METHOD PROTECTED M_DbAlarms : STRING(255)
VAR_INPUT
	nSQLErrorCode				: UDINT;
END_VAR
CASE DatabaseType OF
E_DatabaseType.eMicrosoftSqlCompact,E_DatabaseType.eMicrosoftSql,E_DatabaseType.eMicrosoftAccess:
	CASE nSQLErrorCode OF
		16#80040E00: M_DbAlarms:='Invalid accessor';
		16#80040E01: M_DbAlarms:='Creating another row would have exceeded the total number of active rows supported by the rowset';
		16#80040E02: M_DbAlarms:='Unable to write with a read-only accessor';
		16#80040E03: M_DbAlarms:='Given values violate the database schema';
		16#80040E04: M_DbAlarms:='Invalid row handle';
		16#80040E05: M_DbAlarms:='An object was open';
		16#80040E06: M_DbAlarms:='Invalid chapter';
		16#80040E07: M_DbAlarms:='A literal value in the command could not be converted to the correct type due to a reason other than data overflow';
		16#80040E08: M_DbAlarms:='Invalid binding info';
		16#80040E09: M_DbAlarms:='Permission denied'; 
		16#80040E0A: M_DbAlarms:='Specified column does not contain bookmarks or chapters';
		16#80040E0B: M_DbAlarms:='Some cost limits were rejected';
		16#80040E0C: M_DbAlarms:='No command has been set for the command object';
		16#80040E0D: M_DbAlarms:='Unable to find a query plan within the given cost limit';
		16#80040E0E: M_DbAlarms:='Invalid bookmark';
		16#80040E0F: M_DbAlarms:='Invalid lock mode';
		16#80040E10: M_DbAlarms:='No value given for one or more required parameters';
		16#80040E11: M_DbAlarms:='Invalid column ID';
		16#80040E12: M_DbAlarms:='Invalid ratio';
		16#80040E13: M_DbAlarms:='Invalid value';
		16#80040E14: M_DbAlarms:='The command contained one or more errors';
		16#80040E15: M_DbAlarms:='The executing command cannot be canceled';
		16#80040E16: M_DbAlarms:='The provider does not support the specified dialect';
		16#80040E17: M_DbAlarms:='A data source with the specified name already exists';
		16#80040E18: M_DbAlarms:='The rowset was builtover a live data feed and cannot be restarted';
		16#80040E19: M_DbAlarms:='No key matching the described characteristics could be found within the current range';
		16#80040E1A: M_DbAlarms:='Ownership of this tree has been given to the provider';
		16#80040E1B: M_DbAlarms:='The provider is unable to determine identity for newly inserted rows';
		16#80040E1C: M_DbAlarms:='No nonzero weights specified for any goals supported, so goal was rejected; current goal was not changed';
		16#80040E1D: M_DbAlarms:='Requested conversion is not supported';
		16#80040E1E: M_DbAlarms:='lRowsOffset would position you past either end of the rowset, regardless of the cRows value specified; cRowsObtained is 0';
		16#80040E1F: M_DbAlarms:='Information was requested for a query, and the query was not set';
		16#80040E20: M_DbAlarms:='Provider called a method from IRowsetNotify in the consumer and NT';
		16#80040E21: M_DbAlarms:='Errors occurred';
		16#80040E22: M_DbAlarms:='A non-NULL controlling IUnknown was specified and the object being created does not support aggregation';
		16#80040E23: M_DbAlarms:='A given HROW referred to a hard- or soft-deleted row';
		16#80040E24: M_DbAlarms:='The rowset does not support fetching backwards';
		16#80040E25: M_DbAlarms:='All HROWs must be released before new ones can be obtained';
		16#80040E26: M_DbAlarms:='One of the specified storage flags was not supported';
		16#80040E27: M_DbAlarms:='The comparison operator was invalid';
		16#80040E28: M_DbAlarms:='The specified status flag was neither DBCOLUMNSTATUS_OK nor DBCOLUMNSTATUS_ISNUL';
		16#80040E29: M_DbAlarms:='The rowset cannot scroll backwards';
		16#80040E2A: M_DbAlarms:='Invalid region handle';
		16#80040E2B: M_DbAlarms:='The specified set of rows was not contiguous to or overlapping the rows in the specified watch region';
		16#80040E2C: M_DbAlarms:='A transition from ALL* to MOVE* or EXTEND* was specified';
		16#80040E2D: M_DbAlarms:='The specified region is not a proper subregion of the region identified by the given watch region handle';
		16#80040E2E: M_DbAlarms:='The provider does not support multi-statement commands';
		16#80040E2F: M_DbAlarms:='A specified value violated the integrity constraints for a column or table';
		16#80040E30: M_DbAlarms:='The given type name was unrecognized';
		16#80040E31: M_DbAlarms:='Execution aborted because a resource limit has been reached; no results have been returned';
		16#80040E32: M_DbAlarms:='Cannot clone a command object whose command tree contains a rowset or rowsets';
		16#80040E33: M_DbAlarms:='Cannot represent the current tree as text';
		16#80040E34: M_DbAlarms:='The specified index already exists';
		16#80040E35: M_DbAlarms:='The specified index does not exist';
		16#80040E36: M_DbAlarms:='The specified index was in use';
		16#80040E37: M_DbAlarms:='The specified table does not exist';
		16#80040E38: M_DbAlarms:='The rowset was using optimistic concurrency and the value of a column has been changed since it was last read';
		16#80040E39: M_DbAlarms:='Errors were detected during the copy';
		16#80040E3A: M_DbAlarms:='A specified precision was invalid';
		16#80040E3B: M_DbAlarms:='A specified scale was invalid';
		16#80040E3C: M_DbAlarms:='Invalid table ID';
		16#80040E3D: M_DbAlarms:='A specified type was invalid';
		16#80040E3E: M_DbAlarms:='A column ID was occurred more than once in the specification';
		16#80040E3F: M_DbAlarms:='The specified table already exists';
		16#80040E40: M_DbAlarms:='The specified table was in use';
		16#80040E41: M_DbAlarms:='The specified locale ID was not supported';
		16#80040E42: M_DbAlarms:='The specified record number is invalid';
		16#80040E43: M_DbAlarms:='Although the bookmark was validly formed, no row could be found to match it';
		16#80040E44: M_DbAlarms:='The value of a property was invalid';
		16#80040E45: M_DbAlarms:='The rowset was not chaptered';
		16#80040E46: M_DbAlarms:='Invalid accessor';
		16#80040E47: M_DbAlarms:='Invalid storage flags';
		16#80040E48: M_DbAlarms:='By-ref accessors are not supported by this provider';
		16#80040E49: M_DbAlarms:='Null accessors are not supported by this provider';
		16#80040E4A: M_DbAlarms:='The command was not prepared';
		16#80040E4B: M_DbAlarms:='The specified accessor was not a parameter accessor';
		16#80040E4C: M_DbAlarms:='The given accessor was write-only';
		16#80040E4D: M_DbAlarms:='Authentication failed';
		16#80040E4E: M_DbAlarms:='The change was canceled during notification; no columns are changed';
		16#80040E4F: M_DbAlarms:='The rowset was single-chaptered and the chapter was not released';
		16#80040E50: M_DbAlarms:='Invalid source handle';
		16#80040E51: M_DbAlarms:='The provider cannot derive parameter info and SetParameterInfo has not been called';
		16#80040E52: M_DbAlarms:='The data source object is already initialized';
		16#80040E53: M_DbAlarms:='The provider does not support this method';
		16#80040E54: M_DbAlarms:='The number of rows with pending changes has exceeded the set limit';
		16#80040E55: M_DbAlarms:='The specified column did not exist';
		16#80040E56: M_DbAlarms:='There are pending changes on a row with a reference count of zero';
		16#80040E57: M_DbAlarms:='A literal value in the command overflowed the range of the type of the associated column';
		16#80040E58: M_DbAlarms:='The supplied HRESULT was invalid';
		16#80040E59: M_DbAlarms:='The supplied LookupID was invalid';
		16#80040E5A: M_DbAlarms:='The supplied DynamicErrorID was invalid';
		16#80040E5B: M_DbAlarms:='Unable to get visible data for a newly-inserted row that has not yet been updated';
		16#80040E5C: M_DbAlarms:='Invalid conversion flag';
		16#80040E5D: M_DbAlarms:='The given parameter name was unrecognized';
		16#80040E5E: M_DbAlarms:='Multiple storage objects can not be open simultaneously';
		16#80040E5F: M_DbAlarms:='The requested filter could not be opened';
		16#80040E60: M_DbAlarms:='The requested order could not be opened';
		16#80040E61: M_DbAlarms:='Bad tuple';
		16#80040E62: M_DbAlarms:='Bad coordinate';
		16#80040E63: M_DbAlarms:='The given axis was not valid for this Dataset';
		16#80040E64: M_DbAlarms:='One or more of the given cell ordinals was invalid';
		16#80040E65: M_DbAlarms:='The supplied columnID was invalid';
		16#80040E67: M_DbAlarms:='The supplied command does not have a DBID (Note: DBID is SQL shorthand for Database ID.)';
		16#80040E68: M_DbAlarms:='The supplied DBID already exists';
		16#80040E69: M_DbAlarms:='The maximum number of Sessions supported by the provider has already been created. The consumer must release one or more currently held Sessions before obtaining a new Session object';
		16#80040E72: M_DbAlarms:='The index ID is invalid';
		16#80040E73: M_DbAlarms:='The initialization string does not conform to specification';
		16#80040E74: M_DbAlarms:='The OLE DB root enumerator did not return any providers that matched an of the SOURCES_TYPEs requested';
		16#80040E75: M_DbAlarms:='The initialization string specifies a provider which does not match the currently active provider.';
		16#80040E76: M_DbAlarms:='The specified DBID is invalid';
		16#80040E6A: M_DbAlarms:='Invalid trustee value';
		16#80040E6B: M_DbAlarms:='The trustee is not for the current data source';
		16#80040E6C: M_DbAlarms:='The trustee does not support memberships/collections';
		16#80040E6D: M_DbAlarms:='The object is invalid or unknown to the provider';
		16#80040E6E: M_DbAlarms:='No owner exists for the object';
		16#80040E6F: M_DbAlarms:='The access entry list supplied is invalid';
		16#80040E70: M_DbAlarms:='The trustee supplied as owner is invalid or unknown to the provider';
		16#80040E71: M_DbAlarms:='The permission supplied in the access entry list is invalid';
		16#80040E77: M_DbAlarms:='The ConstraintType was invalid or not supported by the provider.';
		16#80040E78: M_DbAlarms:='The ConstraintType was not CONSTRAINTTYPE_FOREIGNKEY and cForeignKeyColumns was not zero';
		16#80040E79: M_DbAlarms:='The Deferrability was invalid or the value was not supported by the provider';
		16#80040E80: M_DbAlarms:='The MatchType was invalid or the value was not supported by the provider';
		16#80040E8A: M_DbAlarms:='The UpdateRule or DeleteRule was invalid or the value was not supported by the provider';
		16#80040E8B: M_DbAlarms:='The pConstraintID did not exist in the data source';
		16#80040E8C: M_DbAlarms:='The dwFlags was invalid';
		16#80040E8D: M_DbAlarms:='The rguidColumnType pointed to a GUID that does not match the object type of this column or this column was not set';
		16#80040E8E: M_DbAlarms:='The requested URL was out-of-scope';
		16#80040E90: M_DbAlarms:='The provider could not drop the object';
		16#80040E91: M_DbAlarms:='There is no source row';
		16#80040E92: M_DbAlarms:='The OLE DB object represented by this URL is locked by one or more other processes';
		16#80040E93: M_DbAlarms:='The client requested an object type that is only valid for a collection';
		16#80040E94: M_DbAlarms:='The caller requested write access to a read-only object';
		16#80040E95: M_DbAlarms:='The provider could not connect to the server for this object';
		16#80040E96: M_DbAlarms:='The provider could not connect to the server for this object';
		16#80040E97: M_DbAlarms:='The attempt to bind to the object timed out';
		16#80040E98: M_DbAlarms:='The provider was unable to create an object at this URL because an object named by this URL already exists';
		16#80040E99: M_DbAlarms:='The provider could not drop the object';
		16#80040E9A: M_DbAlarms:='The provider was unable to create an object at this URL because the server was out of physical storage';
		16#00040EC0: M_DbAlarms:='Fetching requested number of rows would have exceeded total number of active rows supported by the rowset';
		16#00040EC1: M_DbAlarms:='One or more column types are incompatible; conversion errors will occur during copying';
		16#00040EC2: M_DbAlarms:='Parameter type information has been overridden by caller';
		16#00040EC3: M_DbAlarms:='Skipped bookmark for deleted or non-member row';
		16#00040EC4: M_DbAlarms:='Errors found in validating tree';
		16#00040EC5: M_DbAlarms:='There are no more rowsets';
		16#00040EC6: M_DbAlarms:='Reached start or end of rowset or chapter';
		16#00040EC7: M_DbAlarms:='The provider re-executed the command';
		16#00040EC8: M_DbAlarms:='Variable data buffer ful';
		16#00040EC9: M_DbAlarms:='There are no more results';
		16#00040ECA: M_DbAlarms:='Server cannot release or downgrade a lock until the end of the transaction';
		16#00040ECB: M_DbAlarms:='Specified weight was not supported or exceeded the supported limit and was set to 0 or the supported limit';
		16#00040ECC: M_DbAlarms:='Consumer is uninterested in receiving further notification calls for this reason';
		16#00040ECD: M_DbAlarms:='Input dialect was ignored and text was returned in different dialect';
		16#00040ECE: M_DbAlarms:='Consumer is uninterested in receiving further notification calls for this phase';
		16#00040ECF: M_DbAlarms:='Consumer is uninterested in receiving further notification calls for this reason';
		16#00040ED0: M_DbAlarms:='The operation is being processed asynchronously';
		16#00040ED1: M_DbAlarms:='In order to reposition to the start of the rowset, the provider had to reexecute the query; either the order of the columns changed or columns were added to or removed from the rowset';
		16#00040ED2: M_DbAlarms:='The method had some errors; errors have been returned in the error array';
		16#00040ED3: M_DbAlarms:='Invalid row handle';
		16#00040ED4: M_DbAlarms:='A given HROW referred to a hard-deleted row';
		16#00040ED5: M_DbAlarms:='The provider was unable to keep track of all the changes; the client must refetch the data associated with the watch region using another method';
		16#00040ED6: M_DbAlarms:='Execution stopped because a resource LIMIT has been reached; results obtained so far have been returned but execution cannot be resumed';
		16#00040ED7: M_DbAlarms:='The bind failed because the provider was unable to satisfy all of the bind flags or properties';
		16#00040ED8: M_DbAlarms:='A lock was upgraded FROM the value specified';
		16#00040ED9: M_DbAlarms:='One OR more properties were changed as allowed BY provider';
		16#00040EDA: M_DbAlarms:='Errors occurred';
		16#00040EDB: M_DbAlarms:='A specified parameter was invalid';
		16#00040EDC: M_DbAlarms:='Updating this row caused more than one row to be updated in the data source';
		16#00040EDD: M_DbAlarms:='The row has no row-specific columns';
	ELSE
		M_DbAlarms:= 'Undefined Microsoft Sql Alarm';
	END_CASE
E_DatabaseType.eMySQL:
	//TODO
E_DatabaseType.eOracle:
	//TODO
E_DatabaseType.eDB2:
	//TODO
E_DatabaseType.ePostgreSQL:
	//TODO
E_DatabaseType.eInterbase:
	//TODO
E_DatabaseType.eXml:
	CASE nSQLErrorCode OF
		1:	M_DbAlarms:='FUNCTION NOT allowed.';
		2:	M_DbAlarms:='XML file could not be read';
		3:	M_DbAlarms:='XML schema could not be read';
		4:	M_DbAlarms:='Syntax error';
		5:	M_DbAlarms:='Table could not be created.';
		6:	M_DbAlarms:='The list OF INSERT VALUES are NOT conform TO the collumn list';
		7:	M_DbAlarms:='Memory OF the PLC structure NOT big enough.';
		8:	M_DbAlarms:='XML file could not be created.';
		9:	M_DbAlarms:='XML database not found.';
		10:	M_DbAlarms:='XML table NOT found.';
	ELSE
		M_DbAlarms:= 'Undefined XML DB Alarm';
	END_CASE
E_DatabaseType.eAscii:
	CASE nSQLErrorCode OF
		1:	M_DbAlarms:='FUNCTION NOT allowed.';
		2:	M_DbAlarms:='Syntax error';
		3:	M_DbAlarms:='File could not be open.';
	ELSE
		M_DbAlarms:= 'Undefined ASCII DB Alarm';
	END_CASE
END_CASE
END_METHOD

METHOD PROTECTED M_DbServerAlarms : STRING
VAR_INPUT
	nErrID				: UDINT;
END_VAR
CASE nErrID OF
	131073: M_DbServerAlarms := 'Microsoft SQL Compact database';
	262145: M_DbServerAlarms := 'Microsoft SQL database';
	524289: M_DbServerAlarms := 'Microsoft Access database';
	1048577: M_DbServerAlarms := 'MySQL database';
	2097153: M_DbServerAlarms := 'Oracle database';
	4194305: M_DbServerAlarms := 'DB2 database';
	8388609: M_DbServerAlarms := 'PostgreSQL database';
	16777217: M_DbServerAlarms := 'Interbase/Firebird database';
	33554433: M_DbServerAlarms := 'NULL values are not allowed';
	33554434: M_DbServerAlarms := 'FB_DBRead selected value is NULL';
	33554435: M_DbServerAlarms := 'DBID is unknown';
	33554436: M_DbServerAlarms := 'ADSDevID is unknown';
	33554437: M_DbServerAlarms := 'No open database connection found for DBID xy';
	33554438: M_DbServerAlarms := 'No open ADS device connection found for ADSDevID xy';
	67108865: M_DbServerAlarms := 'XML database';
	134217729: M_DbServerAlarms := 	'ASCII database';
ELSE
	M_DbServerAlarms := 	'ADS Error';
END_CASE
END_METHOD

METHOD PROTECTED M_OdbcAlarms : STRING
VAR_INPUT
	sSQLState    : STRING(5);
END_VAR
IF sSQLState = '1000' THEN  M_OdbcAlarms:= 'General warning';
ELSIF sSQLState ='1001'	THEN M_OdbcAlarms:= 'Cursor operation conflict';
ELSIF sSQLState ='1002'	THEN M_OdbcAlarms:= 'Disconnect error';
ELSIF sSQLState ='1003'	THEN M_OdbcAlarms:= 'NULL value eliminated in set FUNCTION';
ELSIF sSQLState ='1004'	THEN M_OdbcAlarms:= 'STRING data, right-truncated';
ELSIF sSQLState ='1006'	THEN M_OdbcAlarms:= 'Privilege NOT revoked';
ELSIF sSQLState ='1007'	THEN M_OdbcAlarms:= 'Privilege NOT granted';
ELSIF sSQLState ='01S00' THEN M_OdbcAlarms:= 'Invalid connection STRING attribute';
ELSIF sSQLState ='01S01' THEN M_OdbcAlarms:= 'Error in row';
ELSIF sSQLState ='01S02' THEN M_OdbcAlarms:= 'Option value changed';
ELSIF sSQLState ='01S06' THEN M_OdbcAlarms:= 'Attempt TO fetch before the result set returned the first rowset';
ELSIF sSQLState ='01S07' THEN M_OdbcAlarms:= 'Fractional truncation';
ELSIF sSQLState ='01S08' THEN M_OdbcAlarms:= 'Error saving File DSN';
ELSIF sSQLState ='01S09' THEN M_OdbcAlarms:= 'Invalid keyword';
ELSIF sSQLState ='7001'	THEN M_OdbcAlarms:= 'Wrong number OF parameters';
ELSIF sSQLState ='7002'	THEN M_OdbcAlarms:= 'COUNT field incorrect';
ELSIF sSQLState ='7005'	THEN M_OdbcAlarms:= 'Prepared statement not a cursor-specification';
ELSIF sSQLState ='7006'	THEN M_OdbcAlarms:= 'Restricted data type attribute violation';
ELSIF sSQLState ='7009'	THEN M_OdbcAlarms:= 'Invalid descriptor index';
ELSIF sSQLState ='07S01' THEN M_OdbcAlarms:= 'Invalid use OF default parameter';
ELSIF sSQLState ='8001'	THEN M_OdbcAlarms:= 'Client unable TO establish connection';
ELSIF sSQLState ='8002'	THEN M_OdbcAlarms:= 'Connection name in use';
ELSIF sSQLState ='8003'	THEN M_OdbcAlarms:= 'Connection not open';
ELSIF sSQLState ='8004'	THEN M_OdbcAlarms:= 'Server rejected the connection';
ELSIF sSQLState ='8007'	THEN M_OdbcAlarms:= 'Connection failure during transaction';
ELSIF sSQLState ='08S01' THEN M_OdbcAlarms:= 'Communication link failure';
ELSIF sSQLState ='21S01' THEN M_OdbcAlarms:= 'Insert value list does not match column list';
ELSIF sSQLState ='21S02' THEN M_OdbcAlarms:= 'Degree of derived table does not match column list';
ELSIF sSQLState ='22001' THEN M_OdbcAlarms:= 'String data, right-truncated';
ELSIF sSQLState ='22002' THEN M_OdbcAlarms:= 'Indicator variable required but not supplied';
ELSIF sSQLState ='22003' THEN M_OdbcAlarms:= 'Numeric value out of range';
ELSIF sSQLState ='22007' THEN M_OdbcAlarms:= 'Invalid datetime format';
ELSIF sSQLState ='22008' THEN M_OdbcAlarms:= 'Datetime field overflow';
ELSIF sSQLState ='22012' THEN M_OdbcAlarms:= 'Division by zero';
ELSIF sSQLState ='22015' THEN M_OdbcAlarms:= 'Interval field overflow';
ELSIF sSQLState ='22018' THEN M_OdbcAlarms:= 'Invalid character value for cast specification';
ELSIF sSQLState ='22019' THEN M_OdbcAlarms:= 'Invalid escape character';
ELSIF sSQLState ='22025' THEN M_OdbcAlarms:= 'Invalid escape sequence';
ELSIF sSQLState ='22026' THEN M_OdbcAlarms:= 'String data, length mismatch';
ELSIF sSQLState ='23000' THEN M_OdbcAlarms:= 'Integrity constraint violation';
ELSIF sSQLState ='24000' THEN M_OdbcAlarms:= 'Invalid cursor state';
ELSIF sSQLState ='25000' THEN M_OdbcAlarms:= 'Invalid transaction state';
ELSIF sSQLState ='25S01' THEN M_OdbcAlarms:= 'Transaction state';
ELSIF sSQLState ='25S02' THEN M_OdbcAlarms:= 'Transaction is still active';
ELSIF sSQLState ='25S03' THEN M_OdbcAlarms:= 'Transaction is rolled back';
ELSIF sSQLState ='28000' THEN M_OdbcAlarms:= 'Invalid authorization specification';
ELSIF sSQLState ='34000' THEN M_OdbcAlarms:= 'Invalid cursor name';
ELSIF sSQLState ='3C000' THEN M_OdbcAlarms:= 'Duplicate cursor name';
ELSIF sSQLState ='3D000' THEN M_OdbcAlarms:= 'Invalid catalog name';
ELSIF sSQLState ='3F000' THEN M_OdbcAlarms:= 'Invalid schema name';
ELSIF sSQLState ='40001' THEN M_OdbcAlarms:= 'Serialization failure';
ELSIF sSQLState ='40002' THEN M_OdbcAlarms:= 'Integrity constraint violation';
ELSIF sSQLState ='40003' THEN M_OdbcAlarms:= 'Statement completion unknown';
ELSIF sSQLState ='42000' THEN M_OdbcAlarms:= 'Syntax error or access violation';
ELSIF sSQLState ='42S01' THEN M_OdbcAlarms:= 'Base table or view already exists';
ELSIF sSQLState ='42S02' THEN M_OdbcAlarms:= 'Base table or view not found';
ELSIF sSQLState ='42S11' THEN M_OdbcAlarms:= 'Index already exists';
ELSIF sSQLState ='42S12' THEN M_OdbcAlarms:= 'Index not found';
ELSIF sSQLState ='42S21' THEN M_OdbcAlarms:= 'Column already exists';
ELSIF sSQLState ='42S22' THEN M_OdbcAlarms:= 'Column not found';
ELSIF sSQLState ='44000' THEN M_OdbcAlarms:= 'WITH CHECK OPTION violation';
ELSIF sSQLState ='HY000' THEN M_OdbcAlarms:= 'General error';
ELSIF sSQLState ='HY001' THEN M_OdbcAlarms:= 'Memory allocation error';
ELSIF sSQLState ='HY003' THEN M_OdbcAlarms:= 'Invalid application buffer type';
ELSIF sSQLState ='HY004' THEN M_OdbcAlarms:= 'Invalid SQL data type';
ELSIF sSQLState ='HY007' THEN M_OdbcAlarms:= 'Associated statement is not prepared';
ELSIF sSQLState ='HY008' THEN M_OdbcAlarms:= 'Operation canceled';
ELSIF sSQLState ='HY009' THEN M_OdbcAlarms:= 'Invalid use of null pointer';
ELSIF sSQLState ='HY010' THEN M_OdbcAlarms:= 'Function sequence error';
ELSIF sSQLState ='HY011' THEN M_OdbcAlarms:= 'Attribute cannot be set now';
ELSIF sSQLState ='HY012' THEN M_OdbcAlarms:= 'Invalid transaction operation code';
ELSIF sSQLState ='HY013' THEN M_OdbcAlarms:= 'Memory management error';
ELSIF sSQLState ='HY014' THEN M_OdbcAlarms:= 'Limit on the number of handles exceeded';
ELSIF sSQLState ='HY015' THEN M_OdbcAlarms:= 'No cursor name available';
ELSIF sSQLState ='HY016' THEN M_OdbcAlarms:= 'Cannot modify an implementation row descriptor';
ELSIF sSQLState ='HY017' THEN M_OdbcAlarms:= 'Invalid use of an automatically allocated descriptor handle';
ELSIF sSQLState ='HY018' THEN M_OdbcAlarms:= 'Server declined cancel request';
ELSIF sSQLState ='HY019' THEN M_OdbcAlarms:= 'Non-character and non-binary data sent in pieces';
ELSIF sSQLState ='HY020' THEN M_OdbcAlarms:= 'Attempt to concatenate a null value';
ELSIF sSQLState ='HY021' THEN M_OdbcAlarms:= 'Inconsistent descriptor information';
ELSIF sSQLState ='HY024' THEN M_OdbcAlarms:= 'Invalid attribute value';
ELSIF sSQLState ='HY090' THEN M_OdbcAlarms:= 'Invalid string or buffer length';
ELSIF sSQLState ='HY091' THEN M_OdbcAlarms:= 'Invalid descriptor field identifier';
ELSIF sSQLState ='HY092' THEN M_OdbcAlarms:= 'Invalid attribute/option identifier';
ELSIF sSQLState ='HY095' THEN M_OdbcAlarms:= 'Function type out of range';
ELSIF sSQLState ='HY096' THEN M_OdbcAlarms:= 'Invalid information type';
ELSIF sSQLState ='HY097' THEN M_OdbcAlarms:= 'Column type out of range';
ELSIF sSQLState ='HY098' THEN M_OdbcAlarms:= 'Scope type out of range';
ELSIF sSQLState ='HY099' THEN M_OdbcAlarms:= 'Nullable type out of range';
ELSIF sSQLState ='HY100' THEN M_OdbcAlarms:= 'Uniqueness option type out of range';
ELSIF sSQLState ='HY101' THEN M_OdbcAlarms:= 'Accuracy option type out of range';
ELSIF sSQLState ='HY103' THEN M_OdbcAlarms:= 'Invalid retrieval code';
ELSIF sSQLState ='HY104' THEN M_OdbcAlarms:= 'Invalid precision or scale value';
ELSIF sSQLState ='HY105' THEN M_OdbcAlarms:= 'Invalid parameter type';
ELSIF sSQLState ='HY106' THEN M_OdbcAlarms:= 'Fetch type out of range';
ELSIF sSQLState ='HY107' THEN M_OdbcAlarms:= 'Row value out of range';
ELSIF sSQLState ='HY109' THEN M_OdbcAlarms:= 'Invalid cursor position';
ELSIF sSQLState ='HY110' THEN M_OdbcAlarms:= 'Invalid driver completion';
ELSIF sSQLState ='HY111' THEN M_OdbcAlarms:= 'Invalid bookmark value';
ELSIF sSQLState ='HYC00' THEN M_OdbcAlarms:= 'Optional feature not implemented';
ELSIF sSQLState ='HYT00' THEN M_OdbcAlarms:= 'Timeout expired';
ELSIF sSQLState ='HYT01' THEN M_OdbcAlarms:= 'Connection timeout expired';
ELSIF sSQLState ='IM001' THEN M_OdbcAlarms:= 'Driver does not support this function';
ELSIF sSQLState ='IM002' THEN M_OdbcAlarms:= 'Data source name not found and no default driver specified';
ELSIF sSQLState ='IM003' THEN M_OdbcAlarms:= 'Specified driver could not be loaded';
ELSIF sSQLState ='IM004' THEN M_OdbcAlarms:= 'Driver(s) SQLAllocHandle on SQL_HANDLE_ENV failed';
ELSIF sSQLState ='IM005' THEN M_OdbcAlarms:= 'Driver(s) SQLAllocHandle on SQL_HANDLE_DBC failed';
ELSIF sSQLState ='IM006' THEN M_OdbcAlarms:= 'Driver(s) SQLSetConnectAttr failed';
ELSIF sSQLState ='IM007' THEN M_OdbcAlarms:= 'No data source OR driver specified, dialog prohibited';
ELSIF sSQLState ='IM008' THEN M_OdbcAlarms:= 'Dialog failed';
ELSIF sSQLState ='IM009' THEN M_OdbcAlarms:= 'Unable TO load translation DLL';
ELSIF sSQLState ='IM010' THEN M_OdbcAlarms:= 'Data source name too long';
ELSIF sSQLState ='IM011' THEN M_OdbcAlarms:= 'Driver name too long';
ELSIF sSQLState ='IM012' THEN M_OdbcAlarms:= 'DRIVER keyword syntax error';
ELSIF sSQLState ='IM013' THEN M_OdbcAlarms:= 'Trace file error';
ELSIF sSQLState ='IM014' THEN M_OdbcAlarms:= 'Invalid name OF File DSN';
ELSIF sSQLState ='IM015' THEN M_OdbcAlarms:= 'Corrupt file data source';
END_IF
END_METHOD

{attribute 'monitoring' := 'variable'}
PROPERTY PUBLIC Name : String[15]
GET
Name := _Name;
END_GET
SET
_Name := Name;
END_SET
END_PROPERTY

END_FUNCTION_BLOCK

// Objects/FB_SystemEvent_V4_00/FB_SystemEvent
FUNCTION_BLOCK FINAL FB_SystemEvent EXTENDS FB_EventLogger
VAR_INPUT
	Raise					: BOOL;	     				//Event Raiser
	EventType				: E_EventType;				//Event Type Enum 
	EventEntry				: TcEventEntry;				//Event Entry 
	Arg0					: STRING := '';				//Event Argument {0}
	Arg1					: STRING := '';				//Event Argument {1}
	Arg2					: STRING := '';				//Event Argument {2}
END_VAR
VAR_IN_OUT
	Control					: ST_System;				//Machine Control Instance
END_VAR
VAR           
	_EventTimer_ET			: REAL;						//Event timer elapsed
	_Alarm					: BOOL;						//Device Alarm
	_Warning				: BOOL;						//Device Warning
END_VAR
VAR PERSISTENT
	_AlarmMute				: BOOL;						//Event Mute
	_EventTimer_PT			: REAL;						//Event timer preset time
END_VAR

IF NOT _AlarmMute AND NOT Control.Inputs.AlarmAck.Enabled THEN
	IF Raise THEN
		_EventTimer_ET :=  _EventTimer_ET + Control.SystemTime.ScanTime;
	END_IF
END_IF

CASE EventType OF
	E_EventType.eAlarm:
		M_LogAlarm(Execute:= _EventTimer_ET > _EventTimer_PT , Arg0:= Arg0, Arg1:= Arg1, Arg2:= Arg2, EventEntry:= EventEntry,Clear:= NOT _Alarm, Message:= Control.Outputs.AlarmMessage);
		IF _EventTimer_ET > _EventTimer_PT THEN
			IF NOT Control.Outputs.Alarm THEN 
				Control.Outputs.Alarm := TRUE;
			END_IF		
			_Alarm := TRUE;
		END_IF
	E_EventType.eWarning:
		M_LogWarning(Execute:= _EventTimer_ET > _EventTimer_PT , Arg0:= Arg0, Arg1:= Arg1, Arg2:= Arg2, EventEntry:= EventEntry,Clear := NOT _Warning,Message:= Control.Outputs.WarningMessage);
		IF _EventTimer_ET > _EventTimer_PT THEN
			IF NOT Control.Outputs.Warning THEN 
				Control.Outputs.Warning := TRUE;
			END_IF		
			_Warning := TRUE;
		END_IF
	E_EventType.eAlert:
		M_LogAlert(Execute:= Raise, Arg0:= Arg0, Arg1:= Arg1, Arg2:= Arg2, EventEntry:= EventEntry, Message:= Control.Outputs.AlertMessage);
		IF NOT Control.Outputs.Alert AND Raise THEN
			Control.Outputs.Alert := TRUE;
		END_IF
	E_EventType.eMessage:
		M_LogMessage(Execute:= Raise, Arg0:= Arg0, Arg1:= Arg1, Arg2:= Arg2, EventEntry:= EventEntry);
	ELSE
		RETURN;

END_CASE

IF NOT Raise  OR _AlarmMute OR Control.Inputs.AlarmAck.Enabled THEN
	 _EventTimer_ET := 0;_Alarm := FALSE;_Warning := FALSE;
END_IF

{attribute 'monitoring' := 'variable'}
PROPERTY PUBLIC Alarm : Bool
GET
Alarm := _Alarm;
END_GET
END_PROPERTY

{attribute 'monitoring' := 'variable'}
PROPERTY PUBLIC AlarmMute : BOOL
SET
AlarmMute := _AlarmMute;
END_SET
END_PROPERTY

{attribute 'monitoring' := 'variable'}
PROPERTY PUBLIC EventTimer_ET : real
GET
EventTimer_ET := _EventTimer_ET;
END_GET
END_PROPERTY

{attribute 'monitoring' := 'variable'}
PROPERTY PUBLIC EventTimer_PT : real
GET
EventTimer_PT := _EventTimer_PT;
END_GET
SET
_EventTimer_PT := EventTimer_PT;
END_SET
END_PROPERTY

{attribute 'monitoring' := 'variable'}
PROPERTY PUBLIC Warning : Bool
GET
Warning := _Warning;
END_GET
END_PROPERTY

END_FUNCTION_BLOCK

// Objects/FB_Diagnostics_V4_01/FB_Diagnostics
FUNCTION_BLOCK FINAL FB_Diagnostics EXTENDS FB_EventLogger 
VAR_IN_OUT
	Control				: ST_System;					  //Machine Control Instance
	Trigger				: BOOL;							  //Diagnostic function call interval
END_VAR
VAR_OUTPUT
	ncpuUsage 			: UDINT;						  //CPU Usage
	nlatency 			: UDINT;						  //CPU Latency
	Outputs 			: ARRAY[0..255] OF ST_Diagnostics;//Devices on ECAT Bus
	ControllerID		: ST_DeviceIdentificationEx;	  //IPC Information
	IPAddress			: T_IPv4Addr;					  //IPC ip address
END_VAR                                                   
VAR                                                       
	_Alarm				: BOOL;							  //Device Alarm
	_AlarmNum			: DINT;							  //Device Alarm Number
	_Warning			: BOOL;							  //Device Warning
	_WarningNum			: DINT;							  //Device Warning Number
	_FaultTimer_ET		: REAL;								//Fault timer elapsed
	_r_Trig				: ARRAY[0..9] OF R_TRIG;    	  //Public Rising Edge Triggers
END_VAR                                                   
VAR_STAT                                                  
	_Masterdata			: ARRAY[0..10] OF ST_Masterdata;  //ECAT Master Device Diagnostic Data
	_DeviceFault		: BOOL;							  //Fault for crc count
	_StatusFault		: BOOL;							  //Fault for status
END_VAR
VAR PERSISTENT          	
	_Name					: STRING[40];				  //Name for HMI
	_Description			: STRING[40];				  //Description for HMI
	_AlarmMute				: BOOL;						  //Alarm Mute
	_FaultTimer_PT			: REAL;						  //Fault timer preset time
END_VAR

M_CPU();
M_Masters();
M_Slaves();
M_AlarmMonitor();
M_AlarmReset();
M_WarningMonitor();

{attribute 'monitoring' := 'variable'}
PROPERTY PUBLIC Alarm : Bool
GET
Alarm := _Alarm;
END_GET
END_PROPERTY

{attribute 'monitoring' := 'variable'}
PROPERTY PUBLIC AlarmMute : BOOL
SET
AlarmMute := _AlarmMute;
END_SET
END_PROPERTY

{attribute 'monitoring' := 'variable'}
PROPERTY PUBLIC Description : String[40]
GET
Description := _Description;
END_GET
SET
_Description := Description;
END_SET
END_PROPERTY

METHOD PRIVATE F_DeviceState_to_String : STRING
VAR_INPUT
	DeviceState: BYTE;
END_VAR
CASE (DeviceState AND 16#0F) OF
	1: F_DeviceState_to_String := 'Init';
	2: F_DeviceState_to_String := 'Pre-Operational';
	3: F_DeviceState_to_String := 'Bootstrap';
	4: F_DeviceState_to_String := 'Safe-Operational';
	8: F_DeviceState_to_String := 'Operational'; 
END_CASE
CASE (DeviceState AND 16#F0) OF
	1: F_DeviceState_to_String := Concat(F_DeviceState_to_String,': Statemachine error in the EtherCAT slave');
	2: F_DeviceState_to_String := Concat(F_DeviceState_to_String,': Invalid VendorId, Product Code, RevisionsNo or SerialNo');
	4: F_DeviceState_to_String := Concat(F_DeviceState_to_String,': Error occured while sending initialization commands.');
END_CASE
RETURN;
END_METHOD

METHOD PRIVATE F_LinkState_to_String : STRING
VAR_INPUT
	LinkState: BYTE;
END_VAR
CASE (LinkState AND 16#0F) OF
	0: F_LinkState_to_String := 'Link status ok';
	1: F_LinkState_to_String := 'No communication with the EtherCAT-Slave';
	2: F_LinkState_to_String := concat(concat('Error at port ', INT_TO_STRING(((LinkState AND 16#F0)/16)-1)), '. The port has a link, but no communication is possible.');
	4: F_LinkState_to_String := concat(concat('Missing link at port ', BYTE_TO_STRING(((LinkState AND 16#F0)/16)-1)), '.');
	8: F_LinkState_to_String := concat(concat('Additional link at port ', BYTE_TO_STRING(((LinkState AND 16#F0)/16)-1)), '.'); 
END_CASE
RETURN;
END_METHOD

{attribute 'monitoring' := 'variable'}
PROPERTY PUBLIC FaultTimer_PT : real
GET
FaultTimer_PT := _FaultTimer_PT;
END_GET
SET
_FaultTimer_PT := FaultTimer_PT;
END_SET
END_PROPERTY

METHOD PRIVATE M_AlarmMonitor
VAR
END_VAR
VAR_INST // added by the converter: edge detectors and wires of the graphical bodies
    _w1, _w2, _w3, _w4, _w5 : BOOL;
END_VAR
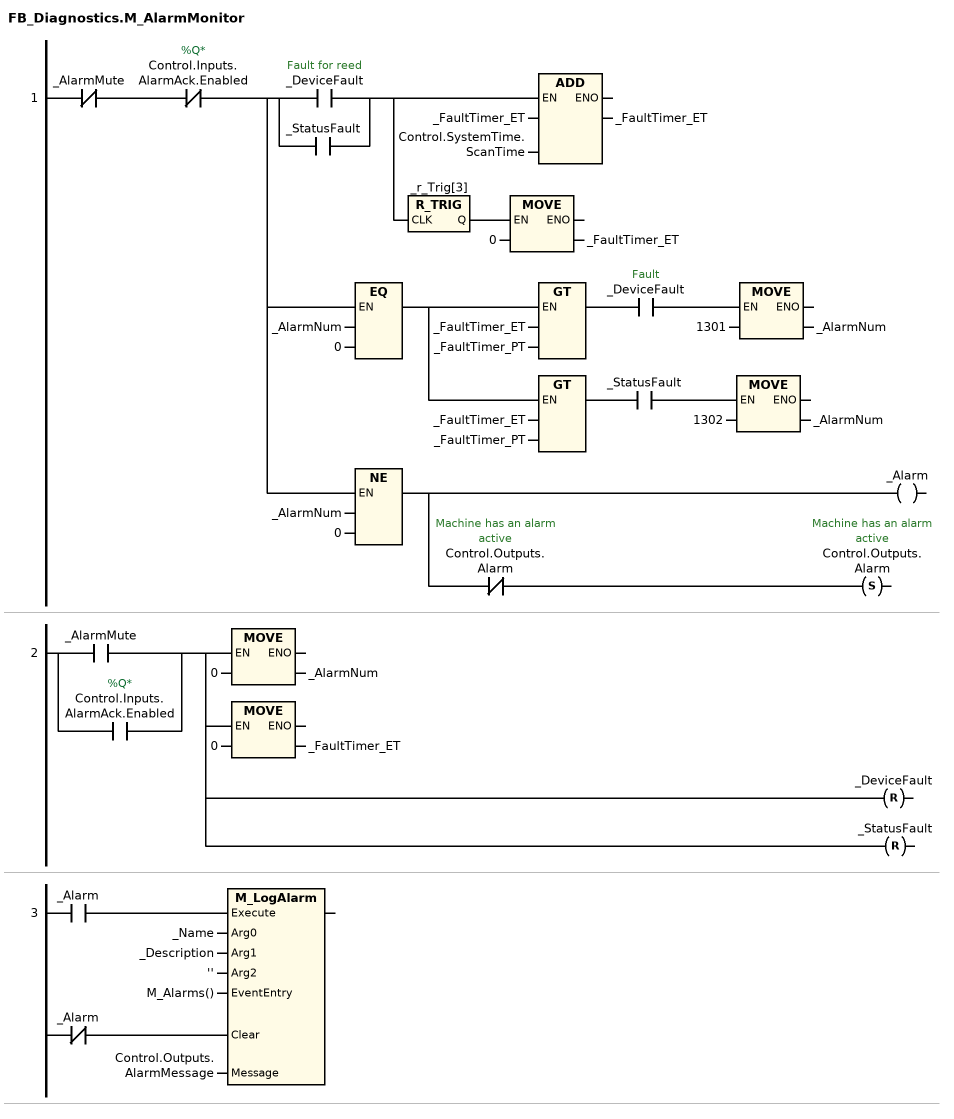
// NETWORK 1
//   Control.Inputs.AlarmAck.Enabled: AT %Q*
//   _DeviceFault: Fault
//   _FaultTimer_ET: Fault timer elapsed
//   Control.SystemTime.ScanTime: Last scan time (Seconds)
//   _FaultTimer_PT: Fault timer preset time
//   Control.Outputs.Alarm: Machine has an alarm active
_w1 := NOT _AlarmMute AND NOT Control.Inputs.AlarmAck.Enabled;
_w2 := _w1 AND (_DeviceFault OR _StatusFault);
IF _w2 THEN _FaultTimer_ET := _FaultTimer_ET + Control.SystemTime.ScanTime; END_IF
_r_Trig[3](CLK := _w2); // R_TRIG
IF _r_Trig[3].Q THEN _FaultTimer_ET := 0; END_IF
_w3 := _w1 AND _AlarmNum = 0;
IF (_w3 AND _FaultTimer_ET > _FaultTimer_PT) AND _DeviceFault THEN _AlarmNum := 1301; END_IF
IF (_w3 AND _FaultTimer_ET > _FaultTimer_PT) AND _StatusFault THEN _AlarmNum := 1302; END_IF
_w4 := _w1 AND _AlarmNum <> 0;
_Alarm := _w4;
Control.Outputs.Alarm S= _w4 AND NOT Control.Outputs.Alarm;

// NETWORK 2
//   Control.Inputs.AlarmAck.Enabled: AT %Q*
//   _FaultTimer_ET: Fault timer elapsed
_w5 := _AlarmMute OR Control.Inputs.AlarmAck.Enabled;
IF _w5 THEN _AlarmNum := 0; END_IF
IF _w5 THEN _FaultTimer_ET := 0; END_IF
_DeviceFault R= _w5;
_StatusFault R= _w5;

// NETWORK 3
M_LogAlarm(Execute := _Alarm, Arg0 := _Name, Arg1 := _Description, Arg2 := '', EventEntry := M_Alarms(), Clear := NOT _Alarm, Message := Control.Outputs.AlarmMessage);
END_METHOD

METHOD PRIVATE M_AlarmReset
VAR_STAT	
	_ClearCRC			:FB_EcMasterFrameStatisticClearCRC; 
	_ClearFrames		:FB_EcMasterFrameStatisticClearFrames;
	_step				: INT;
	_counter			: INT;
END_VAR
// Step engine for resetting etherCat mater errors

CASE _step OF
	0 :	// Initialise and wait for trigger
		_ClearCRC.bExecute:=FALSE;
		_ClearFrames.bExecute:=FALSE;
		_counter := 0;
		IF Control.Inputs.AlarmAck.Enabled THEN _step:=_step+1; END_IF

	
	1 :	// Start getting device ID's 
		_ClearCRC.sNetId := _Masterdata[_counter].NetId;
		_ClearCRC.bExecute:=TRUE;
		IF _ClearCRC.bBusy OR _ClearCRC.bError THEN
		_step:=_step+1; END_IF

	
	2 :	// Getting ID's complete
		_ClearCRC.bExecute:=FALSE;
		IF NOT _ClearCRC.bBusy THEN
		_step:=_step+1;END_IF

	
	3 :	// Start getting device name from device ID
		_ClearFrames.sNetId := _Masterdata[_counter].NetId;
		_ClearFrames.bExecute:=TRUE;
		IF _ClearFrames.bBusy OR _ClearFrames.bError THEN
		_step:=_step+1;END_IF

	
	4 :	// Getting device name complete
		_ClearFrames.bExecute:=FALSE;
		IF NOT _ClearFrames.bBusy THEN
		_step:=_step+1;END_IF

		
	5 :	// Start getting device AMS Net ID from device ID
		_counter := _counter + 1;
		IF _counter >= 11 THEN
		_step:=0;ELSE
		_step:=1;END_IF
			
ELSE
	_step:=0;
END_CASE

// Function block calls
_ClearCRC(sNetId:=);
_ClearFrames(sNetId:=);
END_METHOD

METHOD M_Alarms : TcEventEntry
VAR_INPUT
END_VAR
CASE _AlarmNum OF
	1301: M_Alarms:= TC_Events.TcDiagnostics.A_1301;//Module Fault	
	1302: M_Alarms:= TC_Events.TcDiagnostics.A_1302;//Status Fault			
ELSE
	M_Alarms:= TC_Events.TcDiagnostics.A_Undefined;
END_CASE
END_METHOD

METHOD M_CPU
VAR_STAT
	_DeviceInfo			: FB_GetDeviceIdentificationEx;
	_HostAddr			: FB_GetHostAddrByName;
	_cpuUsage			: TC_CpuUsage;
	_latency			: TC_SysLatency;	
	_incrementer		: INT;	
	_step				: INT;
END_VAR
// Step engine for reading cpu info and status

CASE _step OF
	0 :	// Initialise
		_DeviceInfo.bExecute := FALSE;
		_HostAddr.bExecute := FALSE;
		_cpuUsage.START := FALSE;
		_latency.START := FALSE;
		_step:=_step+1;

	
	1 :	// Start getting device info
		_DeviceInfo.bExecute := TRUE;
		IF _DeviceInfo.bBusy THEN
		_step:=_step+1; END_IF

	
	2 :	// Getting device info completed
		_DeviceInfo.bExecute := FALSE;
		IF NOT _DeviceInfo.bBusy THEN
		_step:=_step+1; END_IF

	
	3 :	// Start getting host AMS address
		_HostAddr.bExecute := TRUE;
		IF _HostAddr.bBusy THEN
		_step:=_step+1; END_IF

	
	4 :	// Getting host AMS address completed
		_HostAddr.bExecute := FALSE;
		IF NOT _HostAddr.bBusy THEN
		_step:=_step+1; END_IF

		
	5 :	// Update outputs
		ControllerID := _DeviceInfo.stDevIdent;
		IPAddress := _HostAddr.sAddr;
		_step:=_step+1;

	
	6 :	// Wait for update trigger
		IF Trigger THEN _step:=_step+1; END_IF

	
	7: 	// Read the cpu usage
		_cpuUsage.START := TRUE;
		IF _cpuUsage.BUSY THEN
		_step:=_step+1; END_IF

		
	8:	// Cpu usage read complete
		_cpuUsage.START := FALSE;
		IF NOT _cpuUsage.BUSY THEN
		_step:=_step+1; END_IF
		
	9:	// Read cpu latency
		_latency.START := TRUE;
		IF _latency.BUSY THEN
		_step:=_step+1; END_IF

		
	10:	// Cpu latency read complete
		_latency.START := FALSE;
		IF NOT _latency.BUSY THEN
		_step:=_step+1; END_IF

		
	11:	// Update outputs and go back to waiting for trigger
		ncpuUsage := _cpuUsage.USAGE;
		nlatency := _latency.ACTUAL;
		_step:=6;
		
ELSE
	_step:=0;
END_CASE

// Function block calls
_DeviceInfo();
_HostAddr(sNetID:=ControllerID.strAmsNetId);
_cpuUsage(NETID:=ControllerID.strAmsNetId);
_latency(NETID:=ControllerID.strAmsNetId);
END_METHOD

METHOD PRIVATE M_Masters
VAR_STAT
	_GetDeviceIDs 				: IOF_GetDeviceIDs;
	_IdsData             		: ARRAY[0..10] OF WORD;	
	_GetDeviceName 				: IOF_GetDeviceName;
	_GetDeviceNetId 			: IOF_GetDeviceNetId;	
	_EcMasterFrameStatistic		: FB_EcMasterFrameStatistic; 
	_GetMasterState    			: FB_EcGetMasterState;
	_step						: INT;
	_counter					: INT;
END_VAR
// Step engine for retrieving etherCat mater info and status
CASE _step OF
	0 :	// Initialise and wait for trigger
		_GetDeviceIDs.START:=FALSE;
		_GetDeviceName.START:=FALSE;
		_GetDeviceNetId.START:=FALSE;
		_EcMasterFrameStatistic.bExecute:=FALSE;
		_GetMasterState.bExecute:=FALSE;
		_counter := 0;
		IF Trigger THEN _step:=_step+1; END_IF
	
	1 :	// Start getting device ID's 
		_GetDeviceIDs.START:=TRUE;
		IF _GetDeviceIDs.BUSY OR _GetDeviceIDs.ERR THEN
		_step:=_step+1; END_IF

	2 :	// Getting ID's complete
		_GetDeviceIDs.START:=FALSE;
		IF NOT _GetDeviceIDs.BUSY THEN
		_step:=_step+1;END_IF
	
	3 :	// Start getting device name from device ID
		_GetDeviceName.DEVICEID := _IdsData[_counter+1];
		_GetDeviceName.START:=TRUE;
		IF _GetDeviceName.BUSY OR _GetDeviceName.ERR THEN
		_step:=_step+1;END_IF
	
	4 :	// Getting device name complete
		_GetDeviceName.START:=FALSE;
		IF NOT _GetDeviceName.BUSY THEN
		_step:=_step+1;END_IF
	
	5 :	// Start getting device AMS Net ID from device ID
		_GetDeviceNetId.DEVICEID := _IdsData[_counter+1];
		_GetDeviceNetId.START:=TRUE;
		IF _GetDeviceNetId.BUSY OR _GetDeviceNetId.ERR THEN
		_step:=_step+1;END_IF
	
	6 :	// Getting device AMS Net ID complete
		_GetDeviceNetId.START:=FALSE;
		IF NOT _GetDeviceNetId.BUSY THEN
		_step:=_step+1;END_IF

	7: 	// Start getting master frame statistics from AMS Net ID
		_EcMasterFrameStatistic.sNetId := _GetDeviceNetId.DeviceNetId;
		_EcMasterFrameStatistic.bExecute := TRUE;
		IF _EcMasterFrameStatistic.bBusy OR _EcMasterFrameStatistic.bError THEN 
		_step := _step+1; END_IF
		
	8:	// Getting frame statistics complete
		_EcMasterFrameStatistic.bExecute:=FALSE;
		IF NOT _EcMasterFrameStatistic.bBusy THEN 
			_step := _step+1; 
		END_IF
	
	9:	// Start getting master status from AMS Net ID
		_GetMasterState.sNetId := _GetDeviceNetId.DeviceNetId;
		_GetMasterState.bExecute := TRUE;
		IF _GetMasterState.bBusy OR _GetMasterState.bError THEN 
		_step := _step+1; END_IF
		
	10:	// Getting master status complete
		IF NOT _GetMasterState.bBusy THEN 
			_GetMasterState.bExecute:=FALSE;
			_step := _step+1; 
		END_IF
	
	11:	// Update master data array
		_Masterdata[_counter].ID := _IdsData[_counter+1];
		_Masterdata[_counter].Name := _GetDeviceName.DEVICENAME;
		_Masterdata[_counter].NetId := _GetDeviceNetId.DeviceNetId;
		_Masterdata[_counter].FramesPerSecond := _EcMasterFrameStatistic.fFramesPerSecond;
		_Masterdata[_counter].LostFrames := _EcMasterFrameStatistic.nLostFrames;
		_Masterdata[_counter].LostQueuedFrames := _EcMasterFrameStatistic.nLostQueuedFrames;
		_Masterdata[_counter].QueuedFramesPerSecond := _EcMasterFrameStatistic.fQueuedFramesPerSecond;
		
		// Convert state word to status text
		IF    _GetMasterState.state = 1 THEN _Masterdata[_counter].Status := 'Init';
		ELSIF _GetMasterState.state = 2 THEN _Masterdata[_counter].Status := 'Pre-Operational';
		ELSIF _GetMasterState.state = 4 THEN _Masterdata[_counter].Status := 'Safe-Operational';
		ELSIF _GetMasterState.state = 8 THEN _Masterdata[_counter].Status := 'Operational';
		ELSE _Masterdata[_counter].Status := 'unknown'; END_IF
		_counter := _counter + 1;
		
		// If another master is in list then retrieve details or return to start and wait for trigger
		IF _IdsData[_counter+1] > 0 THEN
			_step:=3;
		ELSE
			_counter := 0;
			_step:=0;
		END_IF		
ELSE
	_step:=0;
END_CASE

// Function block calls
_GetDeviceIDs(NETID:=,LEN:=SIZEOF(_IdsData),DESTADDR:=ADR(_IdsData));
_GetDeviceName(NETID:=);
_GetDeviceNetId(NETID:=);
_EcMasterFrameStatistic(); 
_GetMasterState();
END_METHOD

METHOD PRIVATE M_Slaves
VAR_STAT
	_step					: INT;
	_counter				: INT;
	_pntr					: INT;
	_MasterCounter			: INT;
	_GetConfSlaves			: FB_EcGetConfSlaves;
	_GetAllSlaveCrcErrors	: FB_EcGetAllSlaveCrcErrors;
	_GetAllSlaveStates		: FB_EcGetAllSlaveStates;
	_crcErrors              : ARRAY[0..255] OF DWORD; 
	_Configs           		: ARRAY[0..255] OF ST_EcSlaveConfigData; 
    _devStates           	: ARRAY[0..255] OF ST_EcSlaveState; 
END_VAR
// Step engine to retrieve etherCat slave device info and status
CASE _step OF
	0 :	// Initialise and wait for trigger
		_GetConfSlaves.bExecute:= FALSE;
		_GetAllSlaveStates.bExecute:= FALSE;
		_GetAllSlaveCrcErrors.bExecute:= FALSE;
		_pntr := 0;
		_counter := 0;
		_MasterCounter := 0;
		IF Trigger THEN _step:=_step+1; END_IF

	1:	// Get master data for output array
		Outputs[_pntr].Name := _Masterdata[_MasterCounter].Name;
		Outputs[_pntr].Address := _Masterdata[_MasterCounter].ID;
		Outputs[_pntr].LostFrames := _Masterdata[_MasterCounter].LostFrames;
		Outputs[_pntr].FramesPerSecond := _Masterdata[_MasterCounter].FramesPerSecond;
		Outputs[_pntr].LostQueuedFrames := _Masterdata[_MasterCounter].LostQueuedFrames;
		Outputs[_pntr].QueuedFramesPerSecond := _Masterdata[_MasterCounter].QueuedFramesPerSecond;
		Outputs[_pntr].NetId := _Masterdata[_MasterCounter].NetId;
		Outputs[_pntr].DeviceStatus := _Masterdata[_MasterCounter].Status;
		_pntr := _pntr + 1;
		
		// Set device and status alarms
		IF _GetAllSlaveStates.nSlaves > 0 THEN
			IF Outputs[_pntr].LostQueuedFrames > 0 OR Outputs[_pntr].LostFrames > 0THEN 
				_Name := Outputs[_pntr].Name;
				_Description := concat(concat('Lost ',UDINT_TO_STRING(Outputs[_pntr].LostFrames + Outputs[_pntr].LostQueuedFrames)),' frames.');
				_DeviceFault := TRUE;
			END_IF
			IF Outputs[_pntr].DeviceStatus <> 'Operational' THEN
				_Name := Outputs[_pntr].Name;
				_Description := Outputs[_pntr].DeviceStatus;
				_StatusFault := TRUE; 
			END_IF
		END_IF
		
		_step:=_step+1;
	2:	// Start getting slave configurations for selected master
		_GetConfSlaves.sNetId:=_Masterdata[_MasterCounter].NetId;
		_GetConfSlaves.bExecute:= TRUE;
		IF _GetConfSlaves.bBusy OR _GetConfSlaves.bError THEN
		_step:=_step+1; END_IF

	3:	// Getting slave configurations complete
		_GetConfSlaves.bExecute:= FALSE;
		IF NOT _GetConfSlaves.bBusy THEN
		_step:=_step+1; END_IF
	
	4:	// Start getting slave crc errors for selected master
		_GetAllSlaveCrcErrors.sNetId:=_Masterdata[_MasterCounter].NetId;
		_GetAllSlaveCrcErrors.bExecute:= TRUE;
		IF _GetAllSlaveCrcErrors.bBusy OR _GetAllSlaveCrcErrors.bError THEN
		_step:=_step+1; END_IF

	
	5:	// Getting slave crc errors complete
		_GetAllSlaveCrcErrors.bExecute:= FALSE;
		IF NOT _GetAllSlaveCrcErrors.bBusy THEN
		_step:=_step+1; END_IF

	6: 	// Start getting slave states for selected master
		_GetAllSlaveStates.sNetId:=_Masterdata[_MasterCounter].NetId;
		_GetAllSlaveStates.bExecute:= TRUE;
		IF _GetAllSlaveStates.bBusy OR _GetAllSlaveStates.bError THEN
		_step:=_step+1; END_IF

	7:	// Getting slave states complete
		_GetAllSlaveStates.bExecute:= FALSE;
		IF NOT _GetAllSlaveStates.bBusy THEN
		_step:=_step+1; END_IF
	
	8:	// Update output array with all slaves for selected master
		IF _GetAllSlaveStates.nSlaves > 0 THEN
			FOR _counter := 0 TO UINT_TO_INT(_GetAllSlaveStates.nSlaves-1) BY 1 DO
				
				Outputs[_pntr].Name := _Configs[_counter].sName;
				Outputs[_pntr].ProductType := _Configs[_counter].sType;
				Outputs[_pntr].CRCError := _crcErrors[_counter];
				Outputs[_pntr].Address := _Configs[_counter].nAddr;
				Outputs[_pntr].LinkStatus := F_LinkState_to_String(_Configs[_counter].nLinkStatus);
				Outputs[_pntr].DeviceStatus := F_DeviceState_to_String(_devStates[_counter].deviceState);
				Outputs[_pntr].NetId := '';
				
				// Set device and status alarms
				IF Outputs[_pntr].CRCError > 0 THEN 
					_Name := Outputs[_pntr].Name;
					_Description := concat(DWORD_TO_STRING(Outputs[_pntr].CRCError),' CRC Errors.');
					_DeviceFault := TRUE; 
				END_IF
				IF Outputs[_pntr].DeviceStatus <> 'Operational' OR Outputs[_pntr].LinkStatus <> 'Link status ok' THEN 
					_Name := Outputs[_pntr].Name;
					_Description := Outputs[_pntr].DeviceStatus;
					_StatusFault := TRUE; 
				END_IF
				
				_pntr := _pntr + 1;
				
			END_FOR
		END_IF
		_step:=_step+1;
	
	9:	// Check if another master in cue and repeat sequence or step forward
		_MasterCounter:=_MasterCounter+1;
		IF _Masterdata[_MasterCounter].Name = '' THEN
		_step:=_step+1; ELSE _step:=1; END_IF	
	
	10:	// Clear the remainder of the output array
		FOR _counter := _pntr TO 255 BY 1 DO
			
			Outputs[_counter].Name := '';
			Outputs[_counter].ProductType := '';
			Outputs[_counter].CRCError := 0;
			Outputs[_counter].Address := 0;
			Outputs[_counter].LinkStatus := '';
			Outputs[_counter].DeviceStatus := '';
			
		END_FOR
		_step:=0;
		
ELSE
	_step:=0;
END_CASE

// Function block calls
_GetConfSlaves(pArrEcConfSlaveInfo := ADR(_Configs), cbBufLen:= SIZEOF(_Configs));
_GetAllSlaveStates(pStateBuf := ADR(_devStates), cbBufLen:=SIZEOF(_devStates));
_GetAllSlaveCrcErrors(pCrcErrorBuf := ADR(_crcErrors), cbBufLen:= SIZEOF(_crcErrors));
END_METHOD

METHOD PRIVATE M_WarningMonitor
VAR_INPUT
END_VAR
VAR_INST
END_VAR
VAR_INST // added by the converter: edge detectors and wires of the graphical bodies
    _w1 : BOOL;
END_VAR
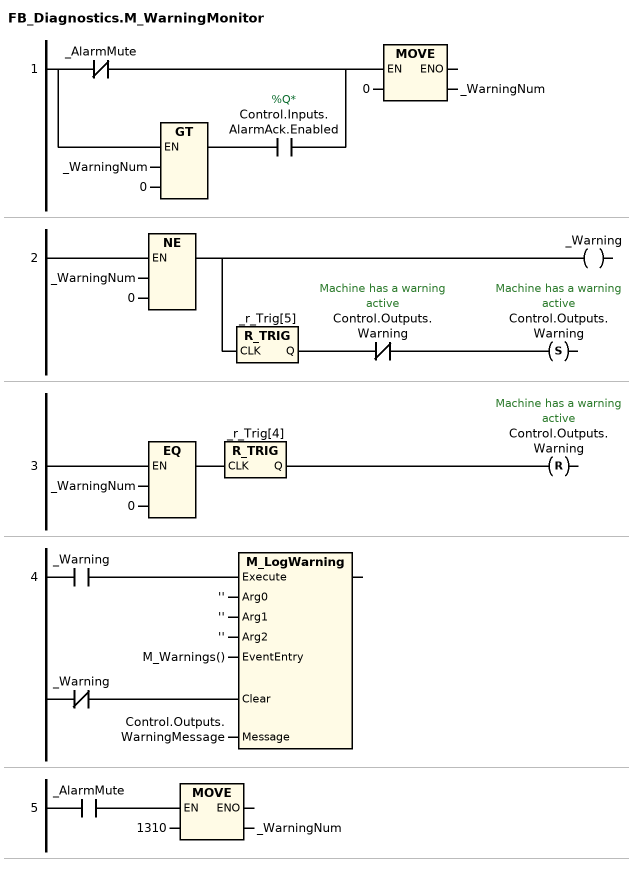
// NETWORK 1
//   Control.Inputs.AlarmAck.Enabled: AT %Q*
IF NOT _AlarmMute OR _WarningNum > 0 AND Control.Inputs.AlarmAck.Enabled THEN _WarningNum := 0; END_IF

// NETWORK 2
//   Control.Outputs.Warning: Machine has a warning active
_w1 := _WarningNum <> 0;
_Warning := _w1;
_r_Trig[5](CLK := _w1); // R_TRIG
Control.Outputs.Warning S= _r_Trig[5].Q AND NOT Control.Outputs.Warning;

// NETWORK 3
//   Control.Outputs.Warning: Machine has a warning active
_r_Trig[4](CLK := _WarningNum = 0); // R_TRIG
Control.Outputs.Warning R= _r_Trig[4].Q;

// NETWORK 4
M_LogWarning(Execute := _Warning, Arg0 := '', Arg1 := '', Arg2 := '', EventEntry := M_Warnings(), Clear := NOT _Warning, Message := Control.Outputs.WarningMessage);

// NETWORK 5
IF _AlarmMute THEN _WarningNum := 1310; END_IF
END_METHOD

METHOD M_Warnings : TcEventEntry
VAR_INPUT
END_VAR
CASE _WarningNum OF
	1310: M_Warnings:= TC_Events.TcDiagnostics.W_1310;//Alarm Mute Active					
ELSE
	M_Warnings:=  TC_Events.TcDiagnostics.W_Undefined;	
END_CASE
END_METHOD

{attribute 'monitoring' := 'variable'}
PROPERTY PUBLIC Name : String[40]
GET
Name := _Name;
END_GET
SET
_Name := Name;
END_SET
END_PROPERTY

{attribute 'monitoring' := 'variable'}
PROPERTY PUBLIC Warning : Bool
GET
Warning := _Warning;
END_GET
END_PROPERTY

END_FUNCTION_BLOCK

// Objects/FB_DolMotor_V4_03/FB_DolMotor
FUNCTION_BLOCK FINAL FB_DolMotor EXTENDS FB_EventLogger 
VAR_INPUT
	Energized					: BOOL;								//Motor Energize Input
	InhibitFeedbackOn			: BOOL;								//Inhibit Feedback On Alarms
	InhibitFeedbackOff			: BOOL;								//Inhibit Feedback Off Alarms
	AutoEN						: BOOL;								//Auto mode enable
END_VAR                                                 			
VAR_IN_OUT                                              			
	Control						: ST_System;						//Machine Control Instance
END_VAR                                                 			
VAR                                                     			
	_AutoFwd					: BOOL;								//Auto of forward command
	_AutoRev					: BOOL;								//Auto of reverse command
	_ManSP1						: BOOL;								//Speed Selection 1
	_ManOnFwd					: BOOL;								//Manual on forwards
	_ManOnRev					: BOOL;								//Manual on reverse
	_ManOff						: BOOL;								//Manual Off
	_ForceOnFwd					: BOOL;								//Force on forward
	_ForceOnRev					: BOOL;								//Force on reverse
	_ForceOff					: BOOL;								//Force off
	_Fault						: BOOL;								//Fault
	_IsolatorFeedback    AT %I*	: BOOL;								//Motor Isolator feedback
	_RunFeedback		 AT %I*	: BOOL;								//Motor Running feedback input
	_OverloadFeedBack    AT %I* : BOOL;								//Motor Overload feedback Input
	_ValueFwd			 AT %Q*	: BOOL;								//Value (physical output)
	_ValueRev			 AT %Q*	: BOOL;								//Value (physical output)
	_ValueSP1			 AT %Q*	: BOOL;								//Value for Secondary Speed (physical output)
	_Velocity			 AT %Q*	: INT;								//Value for Analogue Speed Control (physical output)
	_Running					: BOOL;								//Motor is running
	_MotorOn_ET					: REAL;								//Time output has been on since last being off (sec)
	_FaultTimer_ET				: REAL;								//Fault timer elapsed (sec)
	_Alarm						: BOOL;								//Device Alarm
	_Warning					: BOOL;								//Device Warning
	_AlarmNum					: DINT;								//Device Alarm Number
	_WarningNum					: DINT;								//Device Warning Number
	_R_Trig						: ARRAY[0..9] OF R_TRIG;			//Private Rising Edge Triggers
END_VAR
VAR PERSISTENT
	_Name						: STRING[15];						//Name for HMI
	_Description				: STRING[40];						//Description for HMI
	_AlarmMute					: BOOL;								//Alarm Mute
	_TotalMotorOnHours			: REAL;								//Total Amount of run hours
	_TypeConfig					: SINT;								//0 = DOL Normal, 1 = DOL Reversing
	_StartTimer_PT				: REAL;								//Start Timer Preset
	_FaultTimer_PT				: REAL;								//Fault timer preset time
	_Variables					: ARRAY [0..9] OF ST_Variable;		//Device Associated Varibles Array		
END_VAR

M_AlarmMonitor();
M_WarningMonitor();
M_UnlatchManuals();
M_MotorOutputs();

//Run hours
IF Control.Inputs.HoursReset THEN
	_TotalMotorOnHours := 0;
END_IF
IF _ValueFwd OR _ValueRev THEN
	_MotorOn_ET :=_MotorOn_ET + Control.SystemTime.ScanTime;
ELSE
	_TotalMotorOnHours :=_TotalMotorOnHours + (_MotorOn_ET / 3600);
	_MotorOn_ET := 0;
END_IF

//Motor startup timer
IF (_MotorOn_ET >_StartTimer_PT) THEN
	_Running := TRUE;
ELSE
	_Running := FALSE;
END_IF

{attribute 'monitoring' := 'variable'}
PROPERTY PUBLIC Alarm : Bool
GET
Alarm := _Alarm;
END_GET
END_PROPERTY

{attribute 'monitoring' := 'variable'}
PROPERTY PUBLIC AlarmMute : BOOL
SET
_AlarmMute := AlarmMute;
END_SET
END_PROPERTY

{attribute 'monitoring' := 'variable'}
PROPERTY PUBLIC AutoFwd : BOOL
GET
PUBLIC 
VAR
END_VAR
AutoFwd := _AutoFwd;
END_GET
SET
_AutoFwd := AutoFwd;
END_SET
END_PROPERTY

{attribute 'monitoring' := 'variable'}
PROPERTY PUBLIC AutoRev : BOOL
GET
PUBLIC 
VAR
END_VAR
AutoRev := _AutoRev;
END_GET
SET
_AutoRev := AutoRev;
END_SET
END_PROPERTY

{attribute 'monitoring' := 'variable'}
PROPERTY PUBLIC Description : String[40]
GET
Description := _Description;
END_GET
SET
_Description := Description;
END_SET
END_PROPERTY

{attribute 'monitoring' := 'variable'}
PROPERTY PUBLIC Fault : Bool
SET
_Fault := Fault;
END_SET
END_PROPERTY

{attribute 'monitoring' := 'variable'}
PROPERTY PUBLIC FaultTimer_PT : real
GET
FaultTimer_PT := _FaultTimer_PT;
END_GET
SET
_FaultTimer_PT := FaultTimer_PT;
END_SET
END_PROPERTY

{attribute 'monitoring' := 'variable'}
PROPERTY PUBLIC ForceOff : Bool
GET
ForceOff := _ForceOff;
END_GET
SET
_ForceOff := ForceOff;
END_SET
END_PROPERTY

{attribute 'monitoring' := 'variable'}
PROPERTY PUBLIC ForceOnFwd : Bool
GET
ForceOnFwd := _ForceOnFwd;
END_GET
SET
_ForceOnFwd := ForceOnFwd;
END_SET
END_PROPERTY

{attribute 'monitoring' := 'variable'}
PROPERTY PUBLIC ForceOnRev : Bool
GET
ForceOnRev := _ForceOnRev;
END_GET
SET
_ForceOnRev := ForceOnRev;
END_SET
END_PROPERTY

{attribute 'monitoring' := 'variable'}
PROPERTY PUBLIC IsolatorFeedback : BOOL
GET
PUBLIC 
VAR
END_VAR
IsolatorFeedback := _IsolatorFeedback;
END_GET
SET
_IsolatorFeedback := IsolatorFeedback;
END_SET
END_PROPERTY

METHOD PRIVATE M_AlarmMonitor
VAR_INPUT
END_VAR
VAR_INST
END_VAR
VAR_INST // added by the converter: edge detectors and wires of the graphical bodies
    _w1, _w2, _w3, _w4, _w5 : BOOL;
END_VAR
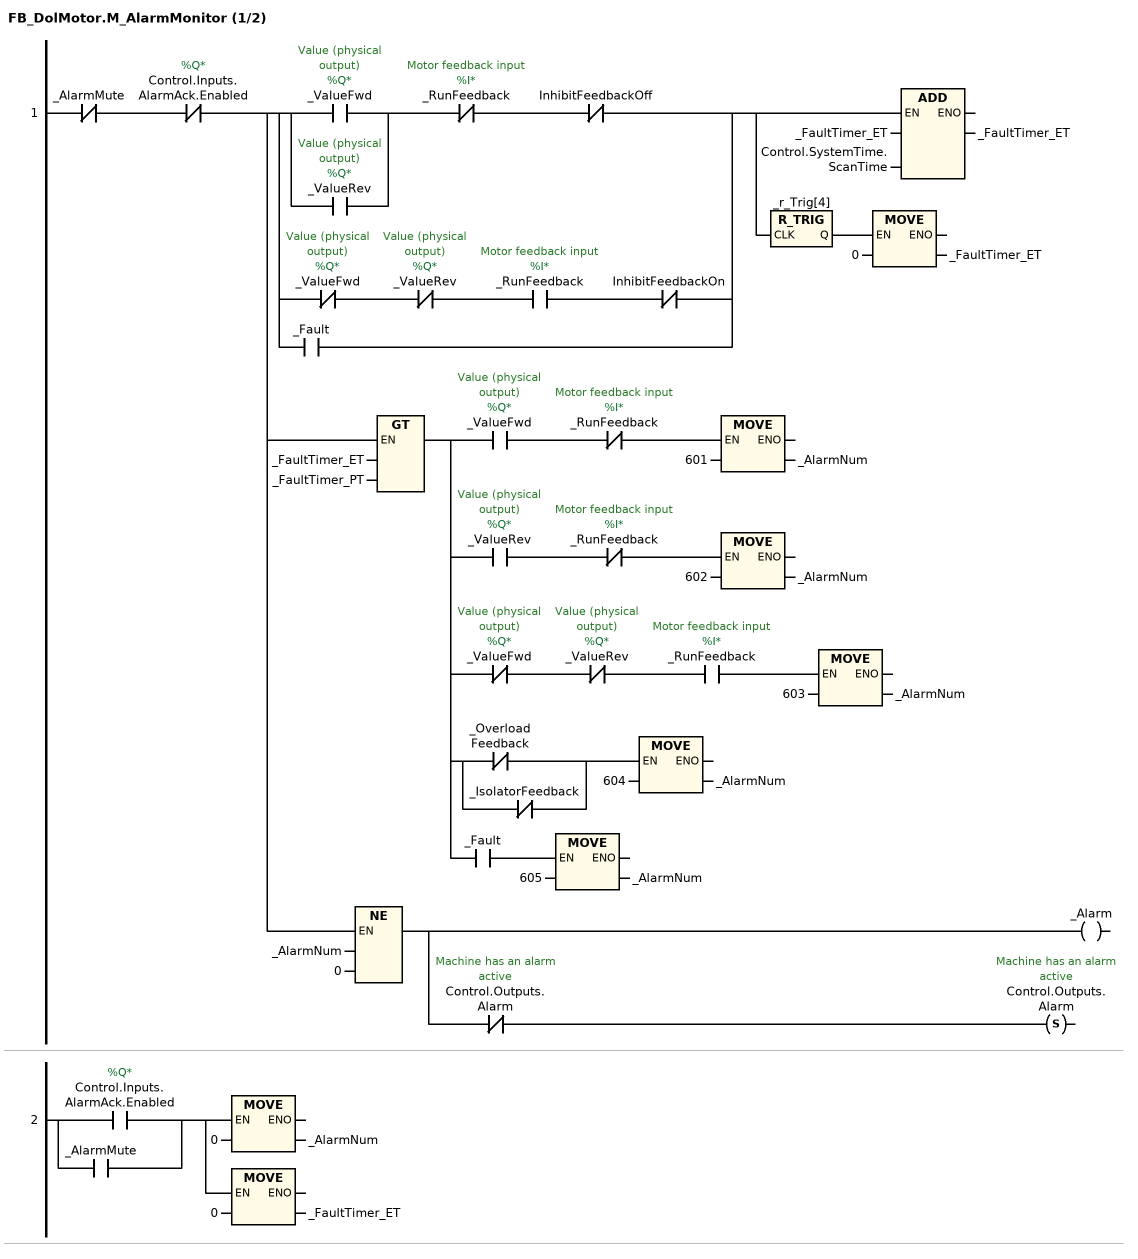
// NETWORK 1
//   Control.Inputs.AlarmAck.Enabled: AT %Q*
//   _ValueFwd: Value (physical output) | AT %Q*
//   _ValueRev: Value (physical output) | AT %Q*
//   _RunFeedback: Motor feedback input | AT %I*
//   _FaultTimer_ET: Fault timer elapsed (sec)
//   Control.SystemTime.ScanTime: Last scan time (Seconds)
//   Control.Outputs.Alarm: Machine has an alarm active
_w1 := NOT _AlarmMute AND NOT Control.Inputs.AlarmAck.Enabled;
_w2 := _w1 AND ((_ValueFwd OR _ValueRev) AND NOT _RunFeedback AND NOT InhibitFeedbackOff OR NOT _ValueFwd AND NOT _ValueRev AND _RunFeedback AND NOT InhibitFeedbackOn OR _Fault);
IF _w2 THEN _FaultTimer_ET := _FaultTimer_ET + Control.SystemTime.ScanTime; END_IF
_r_Trig[4](CLK := _w2); // R_TRIG
IF _r_Trig[4].Q THEN _FaultTimer_ET := 0; END_IF
_w3 := _w1 AND _FaultTimer_ET > _FaultTimer_PT;
IF _w3 AND _ValueFwd AND NOT _RunFeedback THEN _AlarmNum := 601; END_IF
IF _w3 AND _ValueRev AND NOT _RunFeedback THEN _AlarmNum := 602; END_IF
IF _w3 AND NOT _ValueFwd AND NOT _ValueRev AND _RunFeedback THEN _AlarmNum := 603; END_IF
IF _w3 AND (NOT _OverloadFeedback OR NOT _IsolatorFeedback) THEN _AlarmNum := 604; END_IF
IF _w3 AND _Fault THEN _AlarmNum := 605; END_IF
_w4 := _w1 AND _AlarmNum <> 0;
_Alarm := _w4;
Control.Outputs.Alarm S= _w4 AND NOT Control.Outputs.Alarm;

// NETWORK 2
//   Control.Inputs.AlarmAck.Enabled: AT %Q*
//   _FaultTimer_ET: Fault timer elapsed (sec)
_w5 := Control.Inputs.AlarmAck.Enabled OR _AlarmMute;
IF _w5 THEN _AlarmNum := 0; END_IF
IF _w5 THEN _FaultTimer_ET := 0; END_IF

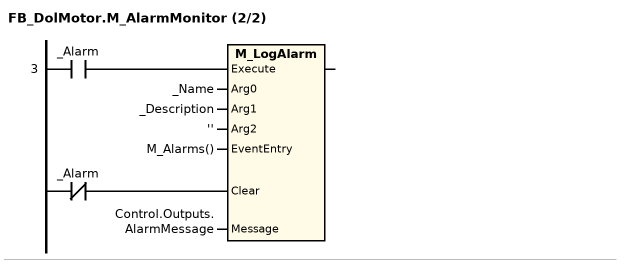
// NETWORK 3
M_LogAlarm(Execute := _Alarm, Arg0 := _Name, Arg1 := _Description, Arg2 := '', EventEntry := M_Alarms(), Clear := NOT _Alarm, Message := Control.Outputs.AlarmMessage);
END_METHOD

METHOD PRIVATE M_Alarms : TcEventEntry
VAR_INPUT
END_VAR
VAR_INST
END_VAR
CASE _AlarmNum OF
601:    M_Alarms :=   TC_Events.TcDolMotor.A_601;//Forward Feedback OFF Alarm
602:    M_Alarms :=   TC_Events.TcDolMotor.A_602;//Reverse Feedback OFF Alarm
603:    M_Alarms :=   TC_Events.TcDolMotor.A_603;//Feedback ON Alarm
604:    M_Alarms :=   TC_Events.TcDolMotor.A_604;//External Feedback Alarm
605:    M_Alarms :=   TC_Events.TcDolMotor.A_605;//Drive Fault
ELSE           
		M_Alarms :=   TC_Events.TcDolMotor.A_Undefined;
END_CASE
END_METHOD

METHOD PRIVATE M_MotorOutputs
VAR_INPUT
END_VAR
VAR_INST
	_Fwd	: BOOL;
	_Rev	: BOOL;
END_VAR
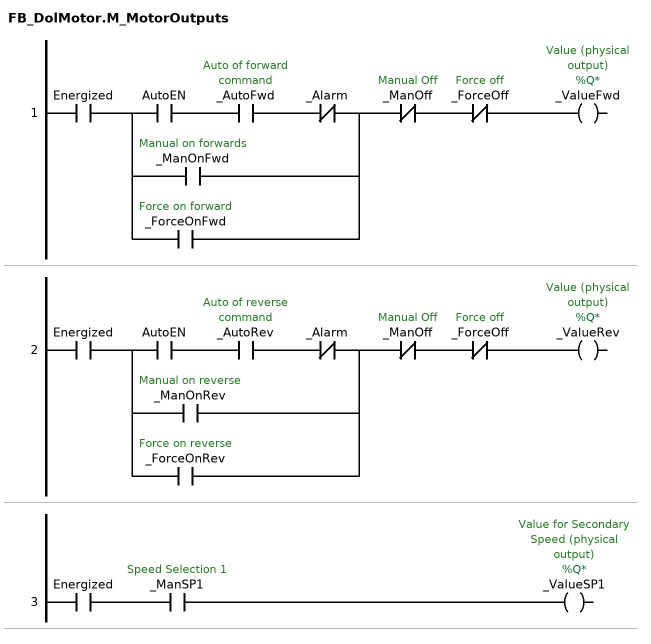
// NETWORK 1
//   _AutoFwd: Auto of forward command
//   _ManOnFwd: Manual on forwards
//   _ForceOnFwd: Force on forward
//   _ManOff: Manual Off
//   _ForceOff: Force off
//   _ValueFwd: Value (physical output) | AT %Q*
_ValueFwd := Energized AND (AutoEN AND _AutoFwd AND NOT _Alarm OR _ManOnFwd OR _ForceOnFwd) AND NOT _ManOff AND NOT _ForceOff;

// NETWORK 2
//   _AutoRev: Auto of reverse command
//   _ManOnRev: Manual on reverse
//   _ForceOnRev: Force on reverse
//   _ManOff: Manual Off
//   _ForceOff: Force off
//   _ValueRev: Value (physical output) | AT %Q*
_ValueRev := Energized AND (AutoEN AND _AutoRev AND NOT _Alarm OR _ManOnRev OR _ForceOnRev) AND NOT _ManOff AND NOT _ForceOff;

// NETWORK 3
//   _ManSP1: Speed Selection 1
//   _ValueSP1: Value for Secondary Speed (physical output) | AT %Q*
_ValueSP1 := Energized AND _ManSP1;
END_METHOD

METHOD PRIVATE M_UnlatchManuals
VAR_INPUT
END_VAR
VAR_INST
END_VAR
VAR_INST // added by the converter: edge detectors and wires of the graphical bodies
    _rt1, _rt2, _rt3, _rt4 : R_TRIG;
END_VAR
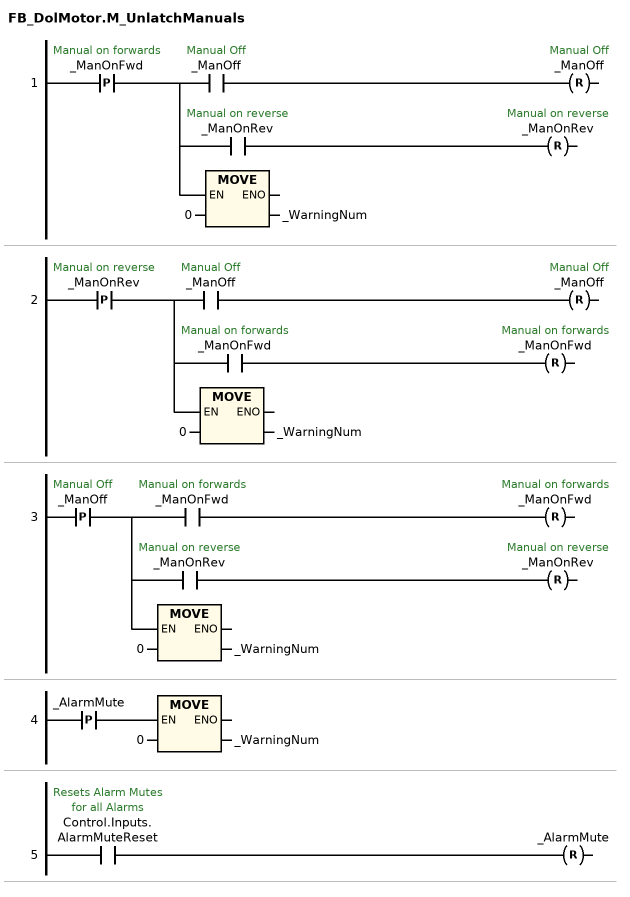
// NETWORK 1
//   _ManOnFwd: Manual on forwards
//   _ManOff: Manual Off
//   _ManOnRev: Manual on reverse
_rt1(CLK := _ManOnFwd);
_ManOff R= _rt1.Q AND _ManOff;
_ManOnRev R= _rt1.Q AND _ManOnRev;
IF _rt1.Q THEN _WarningNum := 0; END_IF

// NETWORK 2
//   _ManOnRev: Manual on reverse
//   _ManOff: Manual Off
//   _ManOnFwd: Manual on forwards
_rt2(CLK := _ManOnRev);
_ManOff R= _rt2.Q AND _ManOff;
_ManOnFwd R= _rt2.Q AND _ManOnFwd;
IF _rt2.Q THEN _WarningNum := 0; END_IF

// NETWORK 3
//   _ManOff: Manual Off
//   _ManOnFwd: Manual on forwards
//   _ManOnRev: Manual on reverse
_rt3(CLK := _ManOff);
_ManOnFwd R= _rt3.Q AND _ManOnFwd;
_ManOnRev R= _rt3.Q AND _ManOnRev;
IF _rt3.Q THEN _WarningNum := 0; END_IF

// NETWORK 4
_rt4(CLK := _AlarmMute);
IF _rt4.Q THEN _WarningNum := 0; END_IF

// NETWORK 5
//   Control.Inputs.AlarmMuteReset: Resets Alarm Mutes for all Alarms
_AlarmMute R= Control.Inputs.AlarmMuteReset;
END_METHOD

METHOD PRIVATE M_WarningMonitor
VAR_INPUT
END_VAR
VAR_INST
END_VAR
VAR_INST // added by the converter: edge detectors and wires of the graphical bodies
    _w1, _w2 : BOOL;
END_VAR
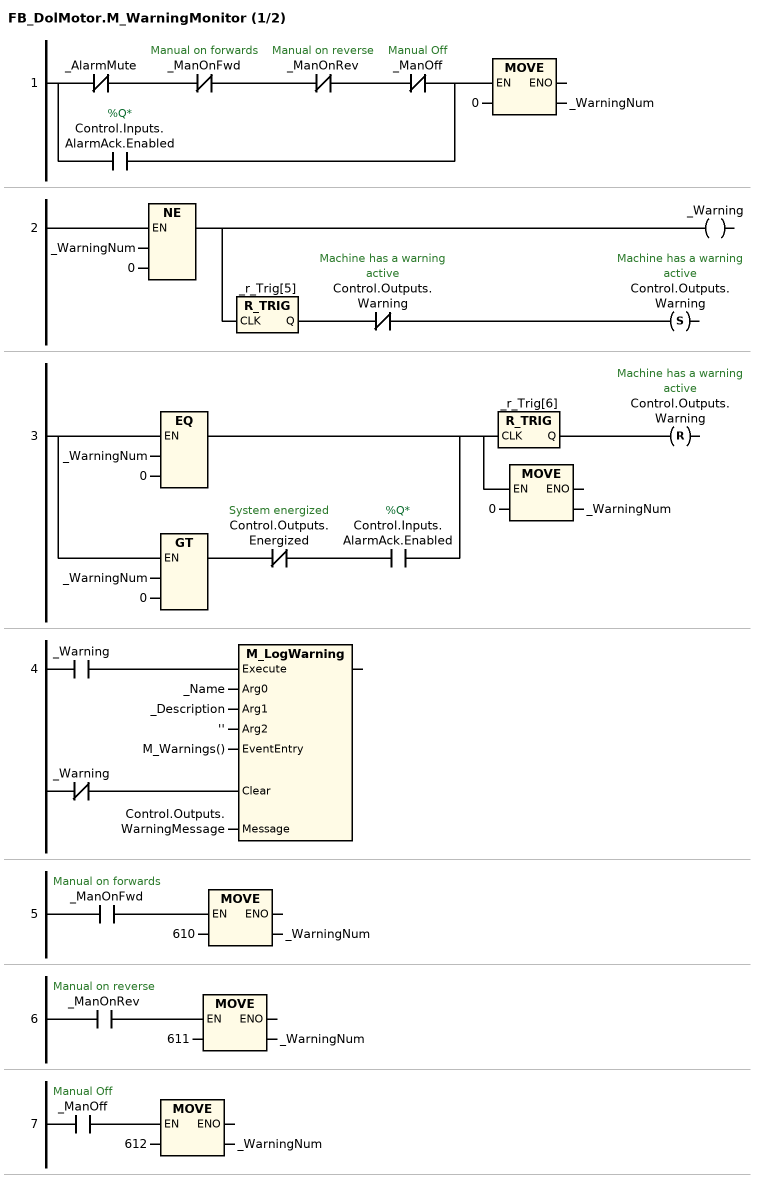
// NETWORK 1
//   _ManOnFwd: Manual on forwards
//   _ManOnRev: Manual on reverse
//   _ManOff: Manual Off
//   Control.Inputs.AlarmAck.Enabled: AT %Q*
IF NOT _AlarmMute AND NOT _ManOnFwd AND NOT _ManOnRev AND NOT _ManOff OR Control.Inputs.AlarmAck.Enabled THEN
    _WarningNum := 0;
END_IF

// NETWORK 2
//   Control.Outputs.Warning: Machine has a warning active
_w1 := _WarningNum <> 0;
_Warning := _w1;
_r_Trig[5](CLK := _w1); // R_TRIG
Control.Outputs.Warning S= _r_Trig[5].Q AND NOT Control.Outputs.Warning;

// NETWORK 3
//   Control.Outputs.Energized: System energized
//   Control.Inputs.AlarmAck.Enabled: AT %Q*
//   Control.Outputs.Warning: Machine has a warning active
_w2 := _WarningNum = 0 OR _WarningNum > 0 AND NOT Control.Outputs.Energized AND Control.Inputs.AlarmAck.Enabled;
_r_Trig[6](CLK := _w2); // R_TRIG
Control.Outputs.Warning R= _r_Trig[6].Q;
IF _w2 THEN _WarningNum := 0; END_IF

// NETWORK 4
M_LogWarning(Execute := _Warning, Arg0 := _Name, Arg1 := _Description, Arg2 := '', EventEntry := M_Warnings(), Clear := NOT _Warning, Message := Control.Outputs.WarningMessage);

// NETWORK 5
//   _ManOnFwd: Manual on forwards
IF _ManOnFwd THEN _WarningNum := 610; END_IF

// NETWORK 6
//   _ManOnRev: Manual on reverse
IF _ManOnRev THEN _WarningNum := 611; END_IF

// NETWORK 7
//   _ManOff: Manual Off
IF _ManOff THEN _WarningNum := 612; END_IF

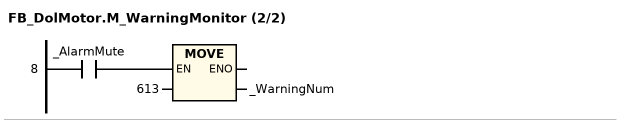
// NETWORK 8
IF _AlarmMute THEN _WarningNum := 613; END_IF
END_METHOD

METHOD PRIVATE M_Warnings : TcEventEntry
VAR_INPUT
END_VAR
VAR_INST
END_VAR
CASE _WarningNum OF
610:    M_Warnings :=   	TC_Events.TcDolMotor.W_610;//Manual ON Enabled
611:    M_Warnings :=   	TC_Events.TcDolMotor.W_611;//Manual Reverse Enabled				
612:    M_Warnings :=   	TC_Events.TcDolMotor.W_612;//Manual OFF Enabled		
613:    M_Warnings :=   	TC_Events.TcDolMotor.W_613;//Alarm Mute Active
ELSE             
		M_Warnings := 	   TC_Events.TcDolMotor.W_Undefined;	
END_CASE
END_METHOD

{attribute 'monitoring' := 'variable'}
PROPERTY PUBLIC ManOff : Bool
GET
ManOff := _ManOff;
END_GET
SET
_ManOff := ManOff;
END_SET
END_PROPERTY

{attribute 'monitoring' := 'variable'}
PROPERTY PUBLIC ManOnFwd : Bool
GET
ManOnFwd := _ManOnFwd;
END_GET
SET
_ManOnFwd := ManOnFwd;
END_SET
END_PROPERTY

{attribute 'monitoring' := 'variable'}
PROPERTY PUBLIC ManOnRev : Bool
GET
ManOnRev := _ManOnRev;
END_GET
SET
_ManOnRev := ManOnRev;
END_SET
END_PROPERTY

{attribute 'monitoring' := 'variable'}
PROPERTY PUBLIC ManSP1 : BOOL
GET
PUBLIC 
VAR
END_VAR
_ManSP1 := ManSP1;
END_GET
SET
_ManSP1 := ManSP1;
END_SET
END_PROPERTY

{attribute 'monitoring' := 'variable'}
PROPERTY PUBLIC MotorOn_ET : real
GET
MotorOn_ET := _MotorOn_ET;
END_GET
END_PROPERTY

{attribute 'monitoring' := 'variable'}
PROPERTY PUBLIC Name : String[15]
GET
Name := _Name;
END_GET
SET
_Name := Name;
END_SET
END_PROPERTY

{attribute 'monitoring' := 'variable'}
PROPERTY PUBLIC OverloadFeedback : BOOL
GET
PUBLIC 
VAR
END_VAR
OverloadFeedback := _OverloadFeedback;
END_GET
SET
_OverloadFeedback := OverloadFeedback;
END_SET
END_PROPERTY

{attribute 'monitoring' := 'variable'}
PROPERTY PUBLIC RunFeedback : BOOL
GET
PUBLIC 
VAR
END_VAR
RunFeedback := _RunFeedback;
END_GET
SET
_RunFeedback := RunFeedback;
END_SET
END_PROPERTY

{attribute 'monitoring' := 'variable'}
PROPERTY PUBLIC Running : Bool
GET
Running := _Running;
END_GET
END_PROPERTY

{attribute 'monitoring' := 'variable'}
PROPERTY PUBLIC StandbyReset : Bool
GET
StandbyReset := _ForceOff;
END_GET
SET
_ForceOff := StandbyReset;
END_SET
END_PROPERTY

{attribute 'monitoring' := 'variable'}
PROPERTY PUBLIC StartTimer_PT : real
GET
StartTimer_PT := _StartTimer_PT;
END_GET
SET
_StartTimer_PT := StartTimer_PT;
END_SET
END_PROPERTY

{attribute 'monitoring' := 'variable'}
PROPERTY PUBLIC TotalMotorOnHours : real
GET
TotalMotorOnHours := _TotalMotorOnHours;
END_GET
END_PROPERTY

{attribute 'monitoring' := 'variable'}
PROPERTY PUBLIC TypeConfig : sint
SET
_TypeConfig := TypeConfig;
END_SET
END_PROPERTY

{attribute 'monitoring' := 'variable'}
PROPERTY PUBLIC ValueFwd : BOOL
GET
PUBLIC 
VAR
END_VAR
ValueFwd := _ValueFwd;
END_GET
SET
_ValueFwd := ValueFwd;
END_SET
END_PROPERTY

{attribute 'monitoring' := 'variable'}
PROPERTY PUBLIC ValueRev : BOOL
GET
PUBLIC 
VAR
END_VAR
ValueRev := _ValueRev;
END_GET
SET
_ValueRev := ValueRev;
END_SET
END_PROPERTY

PROPERTY PUBLIC Variables : REFERENCE TO ARRAY[0..9] OF ST_Variable
GET
Variables REF= _Variables;
END_GET
END_PROPERTY

{attribute 'monitoring' := 'variable'}
PROPERTY PUBLIC Velocity : INT
GET
Velocity:= _Velocity;
END_GET
SET
_Velocity:= Velocity;
END_SET
END_PROPERTY

{attribute 'monitoring' := 'variable'}
PROPERTY PUBLIC Warning : Bool
GET
Warning := _Warning;
END_GET
END_PROPERTY

END_FUNCTION_BLOCK

// Objects/FB_MachineInformation_V4_00/FB_MachineInfo
FUNCTION_BLOCK FB_MachineInfo
VAR_INPUT 
	Trigger				: BOOL;
	RemoveRouteName		: STRING;
	RemoveRoute			: BOOL;
END_VAR
VAR_OUTPUT
	Adapters 			: ARRAY[0..MAX_LOCAL_ADAPTERS] OF ST_IpAdapterInfo;
	Licenses   			: ARRAY[1..nMaxLicenses] OF ST_TcOnlineLicenseInfoData;
	Routes				: ARRAY[0..15] OF ST_AmsRouteEntry;
END_VAR
VAR PERSISTENT
	NetworkDevices 		: ARRAY[0..15] OF ST_IpAdapterInfo;
END_VAR

M_CPU();

METHOD M_CPU
VAR_STAT
	_GetAdaptersInfo	: FB_GetAdaptersInfo;
	_GetLicenses		: FB_GetLicenses;
	_EnumRouteEntry		: FB_EnumRouteEntry;
	_RemoveRouteEntry 	: FB_RemoveRouteEntry;
	_incrementer		: INT;
	_x					: INT;
	_y					: INT;
	_step				: INT;
END_VAR
CASE _step OF
	0 :
		_GetAdaptersInfo.bExecute := FALSE;
		_GetLicenses.bExecute := FALSE;
		_EnumRouteEntry.bExecute := FALSE;
		_EnumRouteEntry.eCmd := eEnumCmd_First;
		_RemoveRouteEntry.bExecute := FALSE;
		_incrementer:=0;
		Trigger:=FALSE;
		_step:=_step+1;

	1 :
		_EnumRouteEntry.bExecute := TRUE;
		IF _EnumRouteEntry.bBusy THEN
		_step:=_step+1; END_IF
	
	2 :
		_EnumRouteEntry.bExecute := FALSE;
		IF NOT _EnumRouteEntry.bBusy THEN
		_step:=_step+1; END_IF
	
	3 :
		IF _EnumRouteEntry.bEOE THEN
			_step:=_step+1; 
			FOR _incrementer := _incrementer TO 15 BY 1 DO
				Routes[_incrementer].dwFlags:=0;
				Routes[_incrementer].eTransport:=0;
				Routes[_incrementer].sAddress:='';
				Routes[_incrementer].sName:='';
				Routes[_incrementer].sNetID:='';
				Routes[_incrementer].tTimeout:=T#0S;
			END_FOR
		ELSE
			Routes[_incrementer]:= _EnumRouteEntry.stRoute;
			_incrementer := _incrementer + 1;
			_EnumRouteEntry.eCmd := eEnumCmd_Next;
			_step:=1;
		END_IF
		
	4 :
		_GetAdaptersInfo.bExecute := TRUE;
		IF _GetAdaptersInfo.bBusy THEN
		_step:=_step+1; END_IF
			
	5 :
		_GetAdaptersInfo.bExecute := FALSE;
		IF NOT _GetAdaptersInfo.bBusy THEN
		_step:=_step+1; END_IF
				
	6 :
		_GetLicenses.bExecute := TRUE;
		IF _GetLicenses.bBusy THEN
		_step:=_step+1; END_IF
				
	7 :
		_GetLicenses.bExecute := FALSE;
		IF NOT _GetLicenses.bBusy THEN
		_step:=_step+1; END_IF
		
	8 :
		Adapters := _GetAdaptersInfo.arrAdapters;
		IF _GetLicenses.nValidLicenses > 0 THEN
			FOR _incrementer := 1 TO UDINT_TO_INT(_GetLicenses.nValidLicenses) DO
				Licenses[_incrementer] := _GetLicenses.aValidLicenses[_incrementer];
			END_FOR
		END_IF
		IF _GetLicenses.nInvalidLicenses > 0 THEN
			FOR _incrementer := UDINT_TO_INT(_GetLicenses.nValidLicenses+1) TO UDINT_TO_INT(_GetLicenses.nValidLicenses + _GetLicenses.nInvalidLicenses) DO
				Licenses[_incrementer] := _GetLicenses.aInvalidLicenses[_incrementer-UDINT_TO_INT(_GetLicenses.nInvalidLicenses)];
			END_FOR
		END_IF
		_step:=_step+1;
		
	9 :
		IF Trigger THEN _step:=0; END_IF
		IF RemoveRoute THEN _step:=_step+1; END_IF
		
	10:
		_RemoveRouteEntry.sName := RemoveRouteName;
		_RemoveRouteEntry.bExecute := TRUE;
		IF _RemoveRouteEntry.bBusy THEN
		_step:=_step+1; END_IF
			
	11:
		_RemoveRouteEntry.bExecute := FALSE;
		IF NOT _RemoveRouteEntry.bBusy THEN
		RemoveRoute := FALSE;
		_step:=0; END_IF
		
ELSE
	_step:=0;
END_CASE

_GetAdaptersInfo();
_GetLicenses();
_EnumRouteEntry();
_RemoveRouteEntry();
END_METHOD

END_FUNCTION_BLOCK

// Objects/FB_MachinePerformance_V4_00/FB_MachinePerformance
FUNCTION_BLOCK FINAL FB_MachinePerformance
VAR_IN_OUT
	Perf										: ARRAY [0..18] OF  ST_Performance_SP;
	Control										: ST_System;
	Data_Reset									: BOOL;
END_VAR
VAR
	_Scratchpad									: DINT;
	_PointerLast								: DINT;
	_Current_Time_T 							: TIME;
	_Current_Time_DT 							: DATE_AND_TIME;
	_Current_Time_TS							: TIMESTRUCT;
	_Today_Time_T								: TIME;
	_Today_Time_DT								: DATE_AND_TIME;
	_Today_Time_TS								: TIMESTRUCT;
	_LifeTime_Time_T							: TIME;
	_LifeTime_Time_DT							: DATE_AND_TIME;
	_LifeTime_Time_TS							: TIMESTRUCT;
	_Perf_Today_Time_T							: TIME;
	_Perf_Today_Time_DT							: DATE_AND_TIME;
	_Perf_Today_Time_TS							: TIMESTRUCT;
	_Perf_LifeTime_Time_T						: TIME;
	_Perf_LifeTime_Time_DT						: DATE_AND_TIME;
	_Perf_LifeTime_Time_TS						: TIMESTRUCT;
	_i											: SINT;
	_j											: SINT;
	_k											: SINT;
END_VAR

IF Control.SystemTime.SecondPulse THEN
	Perf[Control.PackMLState.CurrentState].Current_Time := Perf[Control.PackMLState.CurrentState].Current_Time+1;
	Perf[Control.PackMLState.CurrentState].Today_Time := Perf[Control.PackMLState.CurrentState].Today_Time+1;
	Perf[Control.PackMLState.CurrentState].LifeTime_Time := Perf[Control.PackMLState.CurrentState].LifeTime_Time+1;
	
	_Current_Time_T := DINT_TO_TIME(Perf[Control.PackMLState.CurrentState].Current_Time)*1000;
    _Current_Time_DT := TIME_TO_DT(_Current_Time_T);
    _Current_Time_TS := DT_TO_SYSTEMTIME(_Current_Time_DT);
    IF Perf[Control.PackMLState.CurrentState].Current_Time < 86400 THEN
    	Perf[Control.PackMLState.CurrentState].Current.CurrentTime := MOVE(_Current_Time_TS);
    	Perf[Control.PackMLState.CurrentState].Current.CurrentTime.wDay := 0;
    ELSE
    	Perf[Control.PackMLState.CurrentState].Current.CurrentTime := MOVE(_Current_Time_TS);
    	Perf[Control.PackMLState.CurrentState].Current.CurrentTime.wDay := _Current_Time_TS.wDay-1;
    END_IF	
	
	_Today_Time_T := DINT_TO_TIME(Perf[Control.PackMLState.CurrentState].Today_Time)*1000;
    _Today_Time_DT := TIME_TO_DT(_Today_Time_T);
    _Today_Time_TS := DT_TO_SYSTEMTIME(_Today_Time_DT);
    IF Perf[Control.PackMLState.CurrentState].Today_Time < 86400 THEN
    	Perf[Control.PackMLState.CurrentState].Today.CurrentTime := MOVE(_Today_Time_TS);
    	Perf[Control.PackMLState.CurrentState].Today.CurrentTime.wDay := 0;
    ELSE
    	Perf[Control.PackMLState.CurrentState].Today.CurrentTime := MOVE(_Today_Time_TS);
    	Perf[Control.PackMLState.CurrentState].Today.CurrentTime.wDay := _Today_Time_TS.wDay-1;
    END_IF
	
	_LifeTime_Time_T := DINT_TO_TIME(Perf[Control.PackMLState.CurrentState].LifeTime_Time)*1000;
    _LifeTime_Time_DT := TIME_TO_DT(_LifeTime_Time_T);
    _LifeTime_Time_TS := DT_TO_SYSTEMTIME(_LifeTime_Time_DT);
    IF Perf[Control.PackMLState.CurrentState].LifeTime_Time < 86400 THEN
    	Perf[Control.PackMLState.CurrentState].LifeTime.CurrentTime := MOVE(_LifeTime_Time_TS);
    	Perf[Control.PackMLState.CurrentState].LifeTime.CurrentTime.wDay := 0;
    ELSE
    	Perf[Control.PackMLState.CurrentState].LifeTime.CurrentTime := MOVE(_LifeTime_Time_TS);
    	Perf[Control.PackMLState.CurrentState].LifeTime.CurrentTime.wDay := _LifeTime_Time_TS.wDay-1;
    END_IF	
	
	IF Control.PackMLState.CurrentState <> _PointerLast THEN
		_PointerLast := Control.PackMLState.CurrentState;
		Perf[Control.PackMLState.CurrentState].Today_Freq := Perf[Control.PackMLState.CurrentState].Today_Freq +1;
	END_IF
	
	Perf[0].Today_Time := Perf[1].Today_Time+Perf[2].Today_Time+Perf[3].Today_Time+Perf[4].Today_Time+Perf[5].Today_Time+Perf[6].Today_Time +Perf[7].Today_Time+Perf[8].Today_Time+Perf[9].Today_Time+Perf[10].Today_Time+Perf[11].Today_Time +Perf[12].Today_Time+Perf[13].Today_Time+Perf[14].Today_Time+Perf[15].Today_Time+Perf[16].Today_Time+Perf[17].Today_Time;
	Perf[0].LifeTime_Time := Perf[1].LifeTime_Time+Perf[2].LifeTime_Time+Perf[3].LifeTime_Time+Perf[4].LifeTime_Time+Perf[5].LifeTime_Time+Perf[6].LifeTime_Time+Perf[7].LifeTime_Time+Perf[8].LifeTime_Time+Perf[9].LifeTime_Time+Perf[10].LifeTime_Time+Perf[11].LifeTime_Time+Perf[12].LifeTime_Time+Perf[13].LifeTime_Time+Perf[14].LifeTime_Time+Perf[15].LifeTime_Time+Perf[16].LifeTime_Time+Perf[17].LifeTime_Time;
	
	F_CheckDivDint(Perf[0].LifeTime_Time);
	F_CheckDivDint(Perf[0].Today_Time);
	
	FOR _j:= 1 TO 17 BY 1 DO
		IF Perf[_j].Today_Time > 0 THEN
			Perf[_j].Today_Percent := DINT_TO_REAL((Perf[_j].Today_Time*100)/Perf[0].Today_Time);
		ELSIF Perf[_j].Today_Time = 0 THEN
			Perf[_j].Today_Percent := 0;
		END_IF
		Perf[_j].LifeTime_Percent := DINT_TO_REAL((Perf[_j].LifeTime_Time*100)/Perf[0].LifeTime_Time);
	END_FOR
	
	_Perf_Today_Time_T := DINT_TO_TIME(Perf[0].Today_Time)*1000;
    _Perf_Today_Time_DT := TIME_TO_DT(_Perf_Today_Time_T);
    _Perf_Today_Time_TS := DT_TO_SYSTEMTIME(_Perf_Today_Time_DT);
    IF  Perf[0].Today_Time < 86400 THEN
    	Perf[0].Today.CurrentTime := MOVE(_Current_Time_TS);
    	Perf[0].Today.CurrentTime.wDay := 0;
    ELSE
    	Perf[0].Today.CurrentTime := MOVE(_Current_Time_TS);
    	Perf[0].Today.CurrentTime.wDay := _Current_Time_TS.wDay-1;
    END_IF	
	
	_Perf_LifeTime_Time_T := DINT_TO_TIME(Perf[0].LifeTime_Time)*1000;
    _Perf_LifeTime_Time_DT := TIME_TO_DT(_Perf_LifeTime_Time_T);
    _Perf_LifeTime_Time_TS := DT_TO_SYSTEMTIME(_Perf_LifeTime_Time_DT);
    IF  Perf[0].LifeTime_Time < 86400 THEN
    	Perf[0].LifeTime.CurrentTime := MOVE(_Current_Time_TS);
    	Perf[0].LifeTime.CurrentTime.wDay := 0;
    ELSE
    	Perf[0].LifeTime.CurrentTime := MOVE(_Current_Time_TS);
    	Perf[0].LifeTime.CurrentTime.wDay := _Current_Time_TS.wDay-1;
    END_IF	
	
	F_CheckIndexBounds_DINT(0,17,_Scratchpad);
	FOR _j:= 0 TO 17 BY 1 DO
		IF Perf[_j].Current_Time > 0 AND Control.PackMLState.CurrentState <> _j THEN
			_Scratchpad := 0;
			Perf[_Scratchpad].Current_Time := 0;
			Perf[_Scratchpad].Current.CurrentTime.wDay := 0;
			Perf[_Scratchpad].Current.CurrentTime.wHour:= 0;
			Perf[_Scratchpad].Current.CurrentTime.wMinute := 0;
		END_IF
	END_FOR
END_IF

IF Data_Reset = TRUE THEN
	FOR _k:= 0 TO 17 BY 1 DO
		Perf[_k].Current_Time := 0;
		Perf[_k].Current.CurrentTime.wHour := 0;
		Perf[_k].Current.CurrentTime.wMinute := 0;
		Perf[_k].Current.CurrentTime.wSecond := 0;
		Perf[_k].Today_Time := 0;
		Perf[_k].Today.CurrentTime.wHour := 0;
		Perf[_k].Today.CurrentTime.wMinute := 0;
		Perf[_k].Today.CurrentTime.wSecond := 0;
	END_FOR
END_IF

END_FUNCTION_BLOCK

// Objects/FB_MiscInput_V4_02/FB_MiscInput
FUNCTION_BLOCK FINAL FB_MiscInput EXTENDS FB_EventLogger                                            	
VAR_IN_OUT                                          	
	Control					: ST_System;            	//Machine Control Instance
END_VAR                                             	                                           	
VAR           
	_Input		AT %I*		: BOOL;						//Raw Input 1
	_Input2		AT %I*		: BOOL;						//Raw Input 2                                   	
	_ManOn					: BOOL;	     				//Manual On
	_ManOff					: BOOL;	     				//Manual Off
	_ForceOn				: BOOL;	     				//Force On
	_ForceOff				: BOOL;	     				//Force Off
	_Fault					: BOOL;	     				//Device Fault
	_SimInput				: BOOL;						//Simulates Input
	_FallingEdge			: BOOL;						//Falling Edge of Value Signal
	_RisingEdge				: BOOL;						//Raising Edge of Value Signal
	_DebounceOn_ET			: REAL;						//Debounce On Elapsed Time
	_DebounceOff_ET			: REAL;						//Debounce Off Elapsed Time
	_FaultTimer_ET			: REAL;						//Fault timer elapsed
	_EvaluationError		: BOOL;						//Evaluation Error
	_TestPulseGeneralFault	: BOOL;						//Test Pulse General Fault
	_TestPulse1Fault		: BOOL;						//Test Pulse 1 Fault
	_TestPulse2Fault		: BOOL;						//Test Pulse 2 Fault
	_Alarm					: BOOL;						//Device Alarm
	_Warning				: BOOL;						//Device Warning
	_AlarmNum				: DINT;						//Device Alarm Number
	_WarningNum				: DINT;						//Device Warning Number
	_ConfInput				: BOOL;						//Confirgured Input
	_DebounceOn_DN			: BOOL;						//Debounce On Timer is Done
	_DebounceOff_DN			: BOOL;						//Debounce Off Timer is Done
	_RiseEdge				: R_TRIG;					//Rising Edge Value Trigger
	_FallEdge				: F_TRIG;					//Falling Edge Value Trigger
	_Value		AT %Q*		: BOOL;						//Value of Input
	_R_Trig					: ARRAY[0..9] OF R_TRIG;	//Private Rising Edge Triggers
END_VAR
VAR PERSISTENT
	_Name					: STRING[15];				//Name for HMI
	_Description			: STRING[40];				//Description for HMI
	_AlarmMute				: BOOL;						//Alarm Mute
	_TypeConfig				: E_InputTypeConfig;		//Type congifuration
	_DebounceOn_PT			: REAL;						//Debounce on timer preset time
	_DebounceOff_PT			: REAL;						//Debounce off timer preset time
	_FaultTimer_PT			: REAL;						//Fault timer preset time
END_VAR

M_TypeConfig();
M_AlarmMonitor();
M_WarningMonitor();
M_UnlatchManuals();

//Debounce On Timer
IF _ConfInput = TRUE AND NOT _ForceOff AND NOT _ManOff THEN
	_DebounceOn_ET := _DebounceOn_ET + Control.SystemTime.ScanTime;
	_debounceOn_DN := _DebounceOn_ET > _DebounceOn_PT;
ELSE
	_debounceOn_DN := FALSE;
END_IF
IF _debounceOn_DN OR _ForceOn OR _ManOn THEN
	_Value := TRUE;
	_DebounceOff_ET := 0;
END_IF

//Debounce Off Timer
IF _ConfInput = FALSE AND NOT _ForceOn AND NOT _ManOn THEN
	_DebounceOff_ET := _DebounceOff_ET + Control.SystemTime.ScanTime;
	_debounceOff_DN := _DebounceOff_ET > _DebounceOff_PT;
ELSE
	_debounceOff_DN := FALSE;
END_IF
IF _debounceOff_DN OR _ForceOff OR _ManOff THEN
	_Value := FALSE;
	_DebounceOn_ET := 0;
END_IF

//Rising Edge Trigger 
_riseEdge(CLK := _Value);
_RisingEdge := _riseEdge.Q;

//Falling Edge Trigger
_fallEdge(CLK := _Value);
_FallingEdge := _fallEdge.Q;

{attribute 'monitoring' := 'variable'}
PROPERTY PUBLIC Alarm : Bool
GET
Alarm := _Alarm;
END_GET
END_PROPERTY

{attribute 'monitoring' := 'variable'}
PROPERTY PUBLIC AlarmMute : BOOL
SET
AlarmMute := _AlarmMute;
END_SET
END_PROPERTY

{attribute 'monitoring' := 'variable'}
PROPERTY PUBLIC AutoStandbyReset : Bool
GET
AutoStandbyReset := _ForceOff;
END_GET
SET
_ForceOff := AutoStandbyReset;
END_SET
END_PROPERTY

{attribute 'monitoring' := 'variable'}
PROPERTY PUBLIC DebounceOff_ET : real
GET
DebounceOff_ET := _DebounceOff_ET;
END_GET
END_PROPERTY

{attribute 'monitoring' := 'variable'}
PROPERTY PUBLIC DebounceOff_PT : real
GET
DebounceOff_PT := _DebounceOff_PT;
END_GET
SET
_DebounceOff_PT := DebounceOff_PT;
END_SET
END_PROPERTY

{attribute 'monitoring' := 'variable'}
PROPERTY PUBLIC DebounceOn_ET : real
GET
DebounceOn_ET := _DebounceOn_ET;
END_GET
END_PROPERTY

{attribute 'monitoring' := 'variable'}
PROPERTY PUBLIC DebounceOn_PT : real
GET
DebounceOn_PT := _DebounceOn_PT;
END_GET
SET
_DebounceOn_PT := DebounceOn_PT;
END_SET
END_PROPERTY

{attribute 'monitoring' := 'variable'}
PROPERTY PUBLIC Description : String[40]
GET
Description := _Description;
END_GET
SET
_Description := Description;
END_SET
END_PROPERTY

{attribute 'monitoring' := 'variable'}
PROPERTY PUBLIC EvaluationError : Bool
GET
PUBLIC 
VAR
END_VAR
EvaluationError := _EvaluationError;
END_GET
SET
_EvaluationError := EvaluationError;
END_SET
END_PROPERTY

{attribute 'monitoring' := 'variable'}
PROPERTY PUBLIC FallingEdge : Bool
GET
FallingEdge := _FallingEdge;
END_GET
END_PROPERTY

{attribute 'monitoring' := 'variable'}
PROPERTY PUBLIC Fault : Bool
SET
_Fault := Fault;
END_SET
END_PROPERTY

{attribute 'monitoring' := 'variable'}
PROPERTY PUBLIC FaultTimer_ET : real
GET
FaultTimer_ET := _FaultTimer_ET;
END_GET
END_PROPERTY

{attribute 'monitoring' := 'variable'}
PROPERTY PUBLIC FaultTimer_PT : real
GET
FaultTimer_PT := _FaultTimer_PT;
END_GET
SET
_FaultTimer_PT := FaultTimer_PT;
END_SET
END_PROPERTY

{attribute 'monitoring' := 'variable'}
PROPERTY PUBLIC ForceOn : Bool
GET
ForceOn := _ForceOn;
END_GET
SET
_ForceOn := ForceOn;
END_SET
END_PROPERTY

{attribute 'monitoring' := 'variable'}
PROPERTY PUBLIC Input : Bool
GET
Input := _Input;
END_GET
SET
PUBLIC 
VAR
END_VAR
_Input := Input;
END_SET
END_PROPERTY

{attribute 'monitoring' := 'variable'}
PROPERTY PUBLIC Input2 : Bool
GET
Input2 := _Input2;
END_GET
END_PROPERTY

METHOD PRIVATE M_AlarmMonitor
VAR_IN_OUT
END_VAR
VAR_INST
	_EvaluationError_TON		: 		TON;
END_VAR
VAR_INST // added by the converter: edge detectors and wires of the graphical bodies
    _w1, _w2, _w3, _w4, _w5 : BOOL;
    _rt1 : R_TRIG;
END_VAR
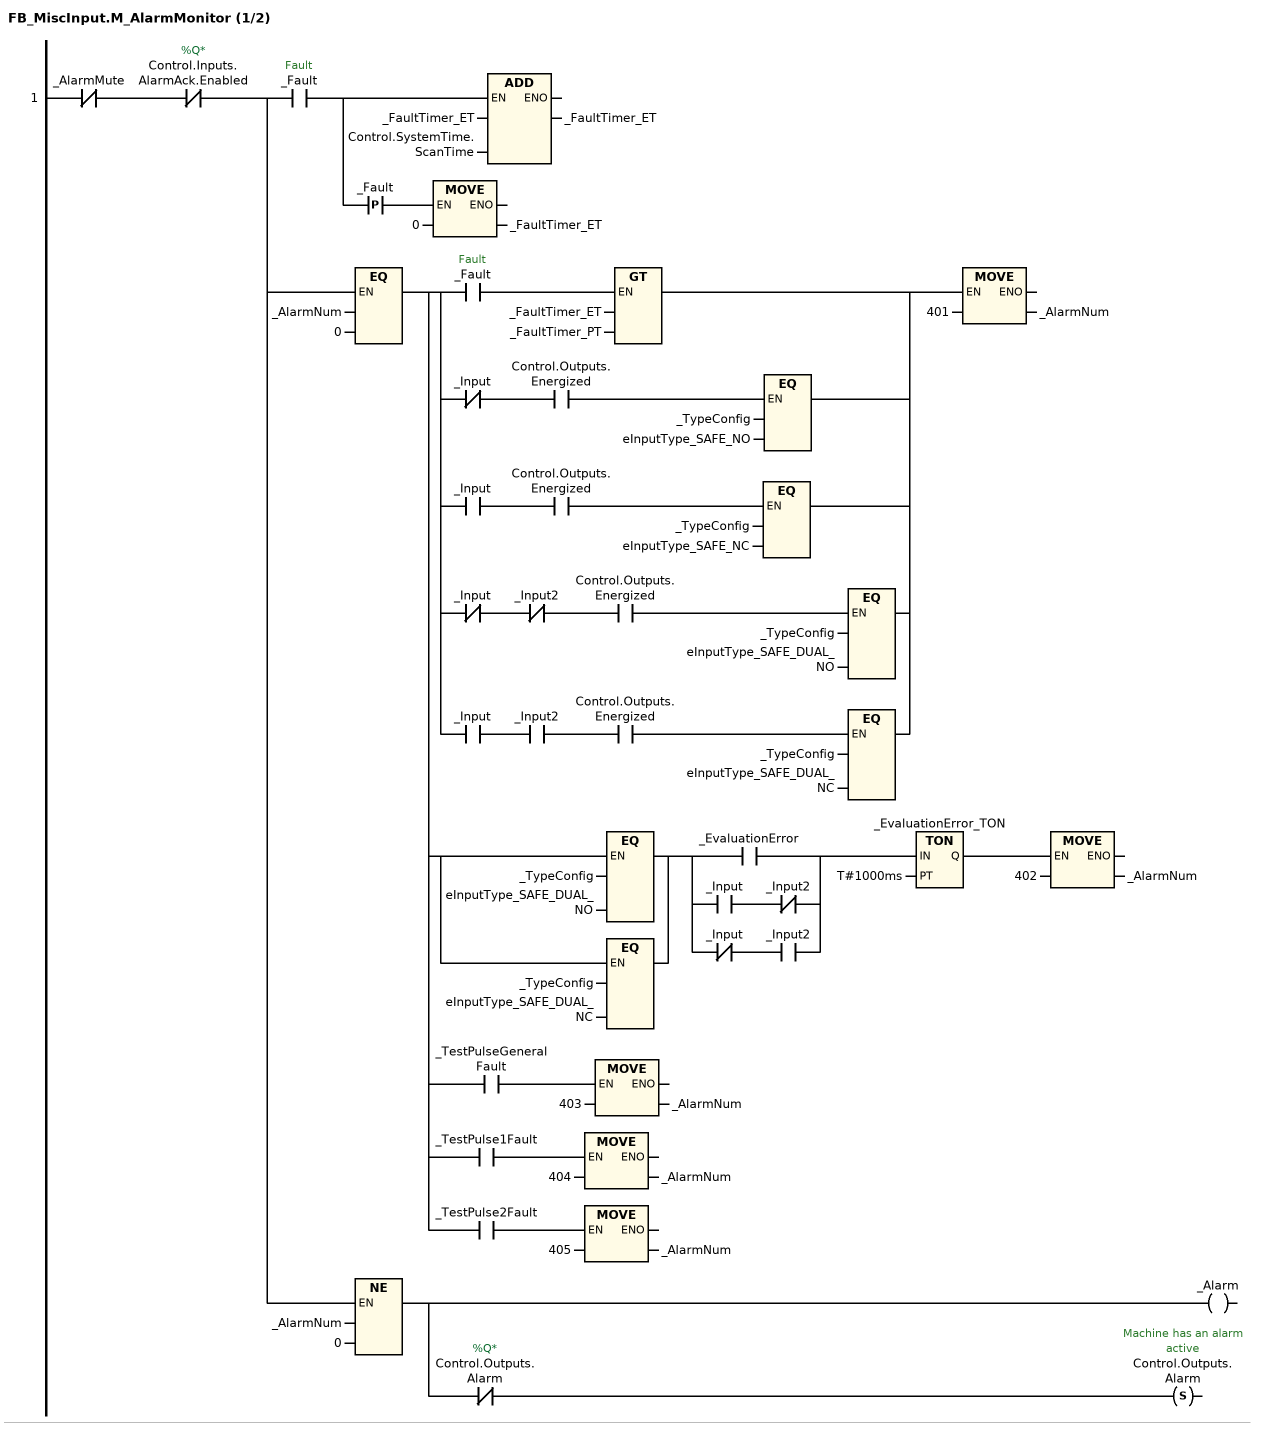
// NETWORK 1
//   Control.Inputs.AlarmAck.Enabled: AT %Q*
//   _Fault: Fault
//   _FaultTimer_ET: Fault timer elapsed
//   Control.SystemTime.ScanTime: Last scan time (Seconds)
//   _FaultTimer_PT: Fault timer preset time
//   Control.Outputs.Alarm: AT %Q* | Machine has an alarm active
_w1 := NOT _AlarmMute AND NOT Control.Inputs.AlarmAck.Enabled;
_w2 := _w1 AND _Fault;
IF _w2 THEN _FaultTimer_ET := _FaultTimer_ET + Control.SystemTime.ScanTime; END_IF
_rt1(CLK := _Fault);
IF _w2 AND _rt1.Q THEN _FaultTimer_ET := 0; END_IF
_w3 := _w1 AND _AlarmNum = 0;
IF _w3 AND _Fault AND _FaultTimer_ET > _FaultTimer_PT OR (_w3 AND NOT _Input) AND Control.Outputs.Energized AND _TypeConfig = eInputType_SAFE_NO OR (_w3 AND _Input) AND Control.Outputs.Energized AND _TypeConfig = eInputType_SAFE_NC OR (_w3 AND NOT _Input) AND NOT _Input2 AND Control.Outputs.Energized AND _TypeConfig = eInputType_SAFE_DUAL_NO OR (_w3 AND _Input) AND _Input2 AND Control.Outputs.Energized AND _TypeConfig = eInputType_SAFE_DUAL_NC THEN
    _AlarmNum := 401;
END_IF
_EvaluationError_TON(IN := (_w3 AND _TypeConfig = eInputType_SAFE_DUAL_NO OR _w3 AND _TypeConfig = eInputType_SAFE_DUAL_NC) AND (_EvaluationError OR _Input AND NOT _Input2 OR NOT _Input AND _Input2), PT := T#1000ms); // TON
IF _EvaluationError_TON.Q THEN _AlarmNum := 402; END_IF
IF _w3 AND _TestPulseGeneralFault THEN _AlarmNum := 403; END_IF
IF _w3 AND _TestPulse1Fault THEN _AlarmNum := 404; END_IF
IF _w3 AND _TestPulse2Fault THEN _AlarmNum := 405; END_IF
_w4 := _w1 AND _AlarmNum <> 0;
_Alarm := _w4;
Control.Outputs.Alarm S= _w4 AND NOT Control.Outputs.Alarm;

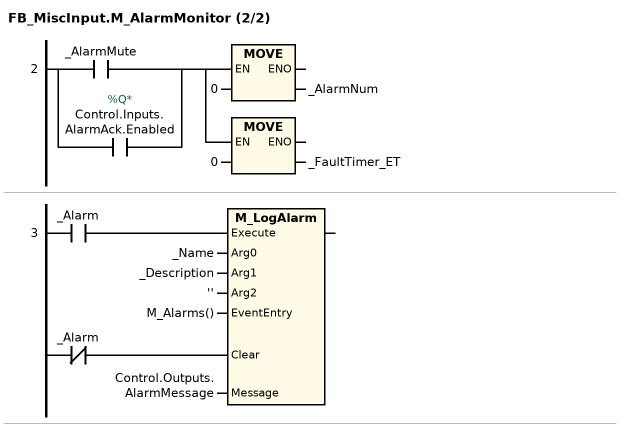
// NETWORK 2
//   Control.Inputs.AlarmAck.Enabled: AT %Q*
//   _FaultTimer_ET: Fault timer elapsed
_w5 := _AlarmMute OR Control.Inputs.AlarmAck.Enabled;
IF _w5 THEN _AlarmNum := 0; END_IF
IF _w5 THEN _FaultTimer_ET := 0; END_IF

// NETWORK 3
M_LogAlarm(Execute := _Alarm, Arg0 := _Name, Arg1 := _Description, Arg2 := '', EventEntry := M_Alarms(), Clear := NOT _Alarm, Message := Control.Outputs.AlarmMessage);
END_METHOD

METHOD PRIVATE M_Alarms : TcEventEntry
VAR_INPUT
END_VAR
CASE _AlarmNum OF
	401: M_Alarms:= TC_Events.TcMiscInput.A_401;//Alarm
	402: M_Alarms:= TC_Events.TcMiscInput.A_402;//Evaluation Error. Contact 1 or 2 failed to switch or switched too late			
	403: M_Alarms:= TC_Events.TcMiscInput.A_403;//Error in the test pulse wiring.
	404: M_Alarms:= TC_Events.TcMiscInput.A_404;//Channel 1 Input Test Pulse Error	
	405: M_Alarms:= TC_Events.TcMiscInput.A_405;//Channel 2 Input Test Pulse Error			
	406: M_Alarms:= TC_Events.TcMiscInput.A_406;//Expected to be ON Fault		
	407: M_Alarms:= TC_Events.TcMiscInput.A_407;//Expected to be OFF Fault						
ELSE
	M_Alarms:= TC_Events.TcMiscInput.A_Undefined;
END_CASE
END_METHOD

METHOD PRIVATE M_TypeConfig
VAR_INPUT
END_VAR
VAR_INST
END_VAR
CASE _TypeConfig OF
	eInputType_PLC_NO, eInputType_SAFE_NO : 
		IF _Input OR _SimInput THEN
			_ConfInput := TRUE;
		ELSE
			_ConfInput := FALSE;
		END_IF
	eInputType_PLC_NC, eInputType_SAFE_NC : 
		IF NOT _Input OR _SimInput THEN
			_ConfInput := TRUE;
		ELSE
			_ConfInput := FALSE;
		END_IF
	eInputType_SAFE_DUAL_NO : 
		IF _Input AND _Input2 THEN
			_ConfInput := TRUE;
		ELSE
			_ConfInput := FALSE;
		END_IF
	eInputType_SAFE_DUAL_NC : 
		IF NOT _Input AND NOT _Input2 THEN
			_ConfInput := TRUE;
		ELSE
			_ConfInput := FALSE;
		END_IF
	eInputType_SAFE_DUAL_NO_NC : 
		IF _Input AND NOT _Input2 THEN
			_ConfInput := TRUE;
		ELSE
			_ConfInput := FALSE;
		END_IF
END_CASE
END_METHOD

METHOD PRIVATE M_UnlatchManuals
VAR_INPUT
END_VAR
VAR_INST
END_VAR
VAR_INST // added by the converter: edge detectors and wires of the graphical bodies
    _rt1, _rt2, _rt3 : R_TRIG;
END_VAR
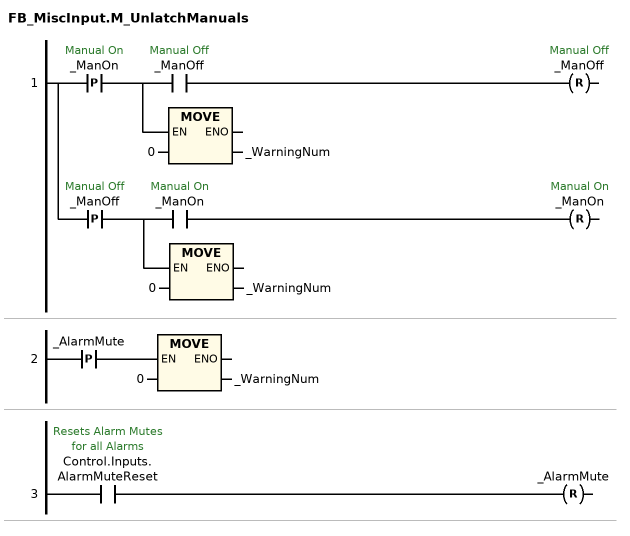
// NETWORK 1
//   _ManOn: Manual On
//   _ManOff: Manual Off
_rt1(CLK := _ManOn);
_ManOff R= _rt1.Q AND _ManOff;
IF _rt1.Q THEN _WarningNum := 0; END_IF
_rt2(CLK := _ManOff);
_ManOn R= _rt2.Q AND _ManOn;
IF _rt2.Q THEN _WarningNum := 0; END_IF

// NETWORK 2
_rt3(CLK := _AlarmMute);
IF _rt3.Q THEN _WarningNum := 0; END_IF

// NETWORK 3
//   Control.Inputs.AlarmMuteReset: Resets Alarm Mutes for all Alarms
_AlarmMute R= Control.Inputs.AlarmMuteReset;
END_METHOD

METHOD PRIVATE M_WarningMonitor
VAR_IN_OUT
END_VAR
VAR_INST
END_VAR
VAR_INST // added by the converter: edge detectors and wires of the graphical bodies
    _w1 : BOOL;
END_VAR
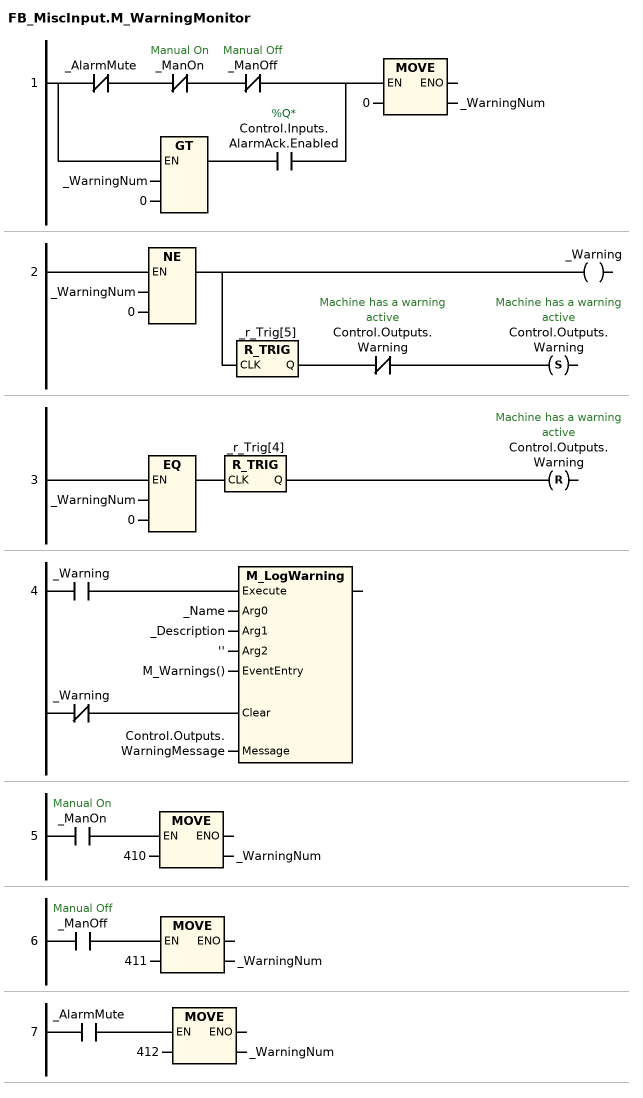
// NETWORK 1
//   _ManOn: Manual On
//   _ManOff: Manual Off
//   Control.Inputs.AlarmAck.Enabled: AT %Q*
IF NOT _AlarmMute AND NOT _ManOn AND NOT _ManOff OR _WarningNum > 0 AND Control.Inputs.AlarmAck.Enabled THEN
    _WarningNum := 0;
END_IF

// NETWORK 2
//   Control.Outputs.Warning: Machine has a warning active
_w1 := _WarningNum <> 0;
_Warning := _w1;
_r_Trig[5](CLK := _w1); // R_TRIG
Control.Outputs.Warning S= _r_Trig[5].Q AND NOT Control.Outputs.Warning;

// NETWORK 3
//   Control.Outputs.Warning: Machine has a warning active
_r_Trig[4](CLK := _WarningNum = 0); // R_TRIG
Control.Outputs.Warning R= _r_Trig[4].Q;

// NETWORK 4
M_LogWarning(Execute := _Warning, Arg0 := _Name, Arg1 := _Description, Arg2 := '', EventEntry := M_Warnings(), Clear := NOT _Warning, Message := Control.Outputs.WarningMessage);

// NETWORK 5
//   _ManOn: Manual On
IF _ManOn THEN _WarningNum := 410; END_IF

// NETWORK 6
//   _ManOff: Manual Off
IF _ManOff THEN _WarningNum := 411; END_IF

// NETWORK 7
IF _AlarmMute THEN _WarningNum := 412; END_IF
END_METHOD

METHOD PRIVATE M_Warnings : TcEventEntry
VAR_INPUT
END_VAR
CASE _WarningNum OF
	410: M_Warnings:= TC_Events.TcMiscInput.W_410;//Manual ON Enabled	
	411: M_Warnings:= TC_Events.TcMiscInput.W_411;//Manual OFF Enabled			
	412: M_Warnings:= TC_Events.TcMiscInput.W_412;//Alarm Mute Active						
ELSE
	M_Warnings:=  TC_Events.TcMiscInput.W_Undefined;
END_CASE
END_METHOD

{attribute 'monitoring' := 'variable'}
PROPERTY PUBLIC ManOff : Bool
GET
ManOff := _ManOff;
END_GET
SET
_ManOff := ManOff;
END_SET
END_PROPERTY

{attribute 'monitoring' := 'variable'}
PROPERTY PUBLIC ManOn : Bool
GET
ManOn := _ManOn;
END_GET
SET
_ManOn := ManOn;
END_SET
END_PROPERTY

{attribute 'monitoring' := 'variable'}
PROPERTY PUBLIC Name : String[15]
GET
Name := _Name;
END_GET
SET
_Name := Name;
END_SET
END_PROPERTY

{attribute 'monitoring' := 'variable'}
PROPERTY PUBLIC RisingEdge : Bool
GET
RisingEdge := _RisingEdge;
END_GET
END_PROPERTY

{attribute 'monitoring' := 'variable'}
PROPERTY PUBLIC SimInput : Bool
SET
_SimInput := SimInput;
END_SET
END_PROPERTY

{attribute 'monitoring' := 'variable'}
PROPERTY PUBLIC TestPulse1Fault : Bool
GET
TestPulse1Fault := _TestPulse1Fault;
END_GET
SET
_TestPulse1Fault := TestPulse1Fault;
END_SET
END_PROPERTY

{attribute 'monitoring' := 'variable'}
PROPERTY PUBLIC TestPulse2Fault : Bool
GET
TestPulse2Fault := _TestPulse2Fault;
END_GET
SET
_TestPulse2Fault := TestPulse2Fault;
END_SET
END_PROPERTY

{attribute 'monitoring' := 'variable'}
PROPERTY PUBLIC TestPulseGeneralFault : Bool
GET
TestPulseGeneralFault := _TestPulseGeneralFault;
END_GET
SET
_TestPulseGeneralFault := TestPulseGeneralFault;
END_SET
END_PROPERTY

{attribute 'monitoring' := 'variable'}
PROPERTY PUBLIC Value : Bool
GET
Value := _Value;
END_GET
SET
_Value := Value;
END_SET
END_PROPERTY

{attribute 'monitoring' := 'variable'}
PROPERTY PUBLIC Warning : Bool
GET
Warning := _Warning;
END_GET
END_PROPERTY

END_FUNCTION_BLOCK

// Objects/FB_MiscOutput_V4_01/FB_MiscOutput
FUNCTION_BLOCK FINAL FB_MiscOutput EXTENDS FB_EventLogger
VAR_INPUT
	Inhibit_Q				: BOOL;						//Inhibit Output
END_VAR                                             	
VAR_IN_OUT                                          	
	Control					: ST_System;            	//Machine Control Instance
END_VAR                                             	
VAR
	_Input		AT %I*		: BOOL;						//Raw Input 1
	_Auto					: BOOL;						//Auto of Output
	_ManOn					: BOOL;						//Manual On
	_ManOff					: BOOL;						//Manual Off
	_ForceOn				: BOOL;						//Force On
	_ForceOff				: BOOL;						//Force Off
	_Fault					: BOOL;						//Device Fault
	_OutputOn_ET			: REAL;						//Time output has been on since last being off
	_OutputOff_ET			: REAL;						//Time output has been off since last being on
	_FaultTimer_ET			: REAL;						//Fault timer elapsed
	_Alarm					: BOOL;						//Device Alarm
	_Warning				: BOOL;						//Device Warning
	_AlarmNum				: DINT;						//Device Alarm Number
	_WarningNum				: DINT;						//Device Warning Number
	_Value			AT %Q*	: BOOL;						//Value (physical output)                                         	
	_R_Trig					: ARRAY[0..9] OF R_TRIG;	//Private Rising Edge Triggers
END_VAR
VAR PERSISTENT
	_Name					: STRING[15];				//Name for HMI
	_Description			: STRING[40];				//Description for HMI
	_AlarmMute				: BOOL;						//Alarm Mute
	_CycleCount				: DINT;						//Total cycles
	_FaultTimer_PT			: REAL;						//Fault timer preset time
END_VAR

M_AlarmMonitor();
M_WarningMonitor();
M_UnlatchManuals();
M_SetOutput();

//Calculate time output has been on/off since last change
IF _Value THEN
	_OutputOn_ET := _OutputOn_ET + Control.SystemTime.ScanTime;
	_OutputOff_ET := 0;
ELSE
	_OutputOff_ET := _OutputOff_ET + Control.SystemTime.ScanTime;
	_OutputOn_ET := 0;
END_IF;

{attribute 'monitoring' := 'variable'}
PROPERTY PUBLIC Alarm : Bool
GET
Alarm := _Alarm;
END_GET
END_PROPERTY

{attribute 'monitoring' := 'variable'}
PROPERTY PUBLIC AlarmMute : BOOL
SET
AlarmMute := _AlarmMute;
END_SET
END_PROPERTY

{attribute 'monitoring' := 'variable'}
PROPERTY PUBLIC Auto : Bool
GET
PUBLIC 
VAR
END_VAR
Auto := _Auto;
END_GET
SET
_Auto := Auto;
END_SET
END_PROPERTY

{attribute 'monitoring' := 'variable'}
PROPERTY PUBLIC CycleCount : DINT
GET
CycleCount := _CycleCount;
END_GET
END_PROPERTY

{attribute 'monitoring' := 'variable'}
PROPERTY PUBLIC Description : String[40]
GET
Description := _Description;
END_GET
SET
_Description := Description;
END_SET
END_PROPERTY

{attribute 'monitoring' := 'variable'}
PROPERTY PUBLIC Fault : Bool
SET
_Fault := Fault;
END_SET
END_PROPERTY

{attribute 'monitoring' := 'variable'}
PROPERTY PUBLIC FaultTimer_ET : real
GET
FaultTimer_ET := _FaultTimer_ET;
END_GET
END_PROPERTY

{attribute 'monitoring' := 'variable'}
PROPERTY PUBLIC FaultTimer_PT : real
GET
FaultTimer_PT := _FaultTimer_PT;
END_GET
SET
_FaultTimer_PT := FaultTimer_PT;
END_SET
END_PROPERTY

{attribute 'monitoring' := 'variable'}
PROPERTY PUBLIC ForceOff : Bool
GET
ForceOff := _ForceOff;
END_GET
SET
_ForceOff := ForceOff;
END_SET
END_PROPERTY

{attribute 'monitoring' := 'variable'}
PROPERTY PUBLIC ForceOn : Bool
GET
ForceOn := _ForceOn;
END_GET
SET
_ForceOn := ForceOn;
END_SET
END_PROPERTY

{attribute 'monitoring' := 'variable'}
PROPERTY PUBLIC Input : Bool
GET
Input := _Input;
END_GET
END_PROPERTY

METHOD PRIVATE M_AlarmMonitor
VAR_INPUT
END_VAR
VAR_INST
END_VAR
VAR_INST // added by the converter: edge detectors and wires of the graphical bodies
    _w1, _w2, _w3 : BOOL;
    _rt1 : R_TRIG;
END_VAR
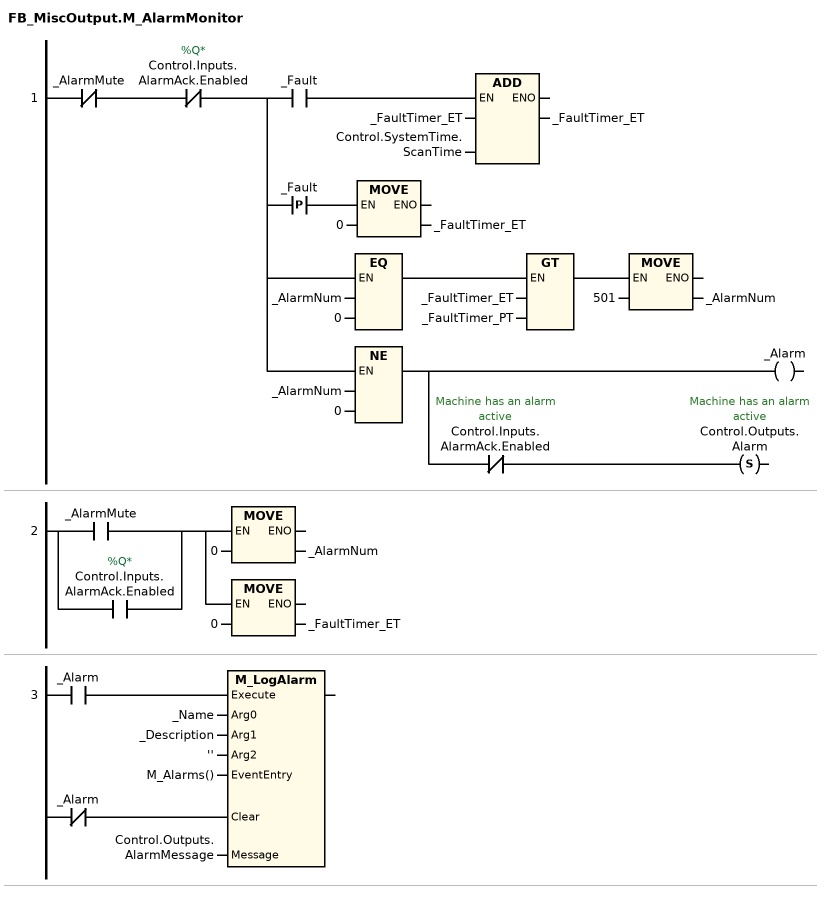
// NETWORK 1
//   Control.Inputs.AlarmAck.Enabled: AT %Q* | Machine has an alarm active
//   _FaultTimer_ET: Fault timer elapsed
//   Control.SystemTime.ScanTime: Last scan time (Seconds)
//   _FaultTimer_PT: Fault timer preset time
//   Control.Outputs.Alarm: Machine has an alarm active
_w1 := NOT _AlarmMute AND NOT Control.Inputs.AlarmAck.Enabled;
IF _w1 AND _Fault THEN _FaultTimer_ET := _FaultTimer_ET + Control.SystemTime.ScanTime; END_IF
_rt1(CLK := _Fault);
IF _w1 AND _rt1.Q THEN _FaultTimer_ET := 0; END_IF
IF _w1 AND _AlarmNum = 0 AND _FaultTimer_ET > _FaultTimer_PT THEN _AlarmNum := 501; END_IF
_w2 := _w1 AND _AlarmNum <> 0;
_Alarm := _w2;
Control.Outputs.Alarm S= _w2 AND NOT Control.Inputs.AlarmAck.Enabled;

// NETWORK 2
//   Control.Inputs.AlarmAck.Enabled: AT %Q*
//   _FaultTimer_ET: Fault timer elapsed
_w3 := _AlarmMute OR Control.Inputs.AlarmAck.Enabled;
IF _w3 THEN _AlarmNum := 0; END_IF
IF _w3 THEN _FaultTimer_ET := 0; END_IF

// NETWORK 3
M_LogAlarm(Execute := _Alarm, Arg0 := _Name, Arg1 := _Description, Arg2 := '', EventEntry := M_Alarms(), Clear := NOT _Alarm, Message := Control.Outputs.AlarmMessage);
END_METHOD

METHOD PRIVATE M_Alarms : TcEventEntry
VAR_INPUT
END_VAR
CASE _AlarmNum OF
	501: M_Alarms:= TC_Events.TcMiscOutput.A_501;//Alarm				
ELSE
	M_Alarms:= TC_Events.TcMiscOutput.A_Undefined;
END_CASE
END_METHOD

METHOD PRIVATE M_SetOutput
VAR
END_VAR
VAR_INST
END_VAR
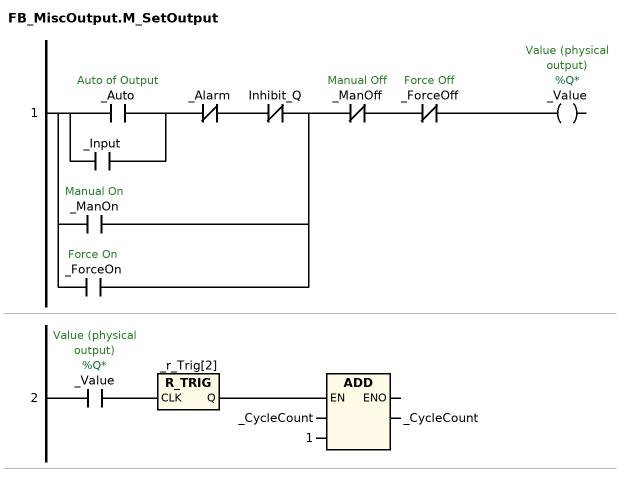
// NETWORK 1
//   _Auto: Auto of Output
//   _ManOn: Manual On
//   _ForceOn: Force On
//   _ManOff: Manual Off
//   _ForceOff: Force Off
//   _Value: Value (physical output) | AT %Q*
_Value := ((_Auto OR _Input) AND NOT _Alarm AND NOT Inhibit_Q OR _ManOn OR _ForceOn) AND NOT _ManOff AND NOT _ForceOff;

// NETWORK 2
//   _Value: Value (physical output) | AT %Q*
//   _CycleCount: Total cycles
_r_Trig[2](CLK := _Value); // R_TRIG
IF _r_Trig[2].Q THEN _CycleCount := _CycleCount + 1; END_IF
END_METHOD

METHOD PRIVATE M_UnlatchManuals
VAR_INPUT
END_VAR
VAR_INST
END_VAR
VAR_INST // added by the converter: edge detectors and wires of the graphical bodies
    _rt1, _rt2, _rt3 : R_TRIG;
END_VAR
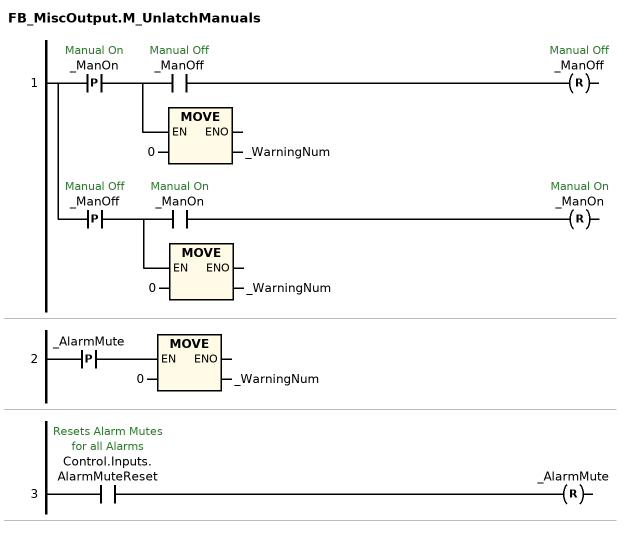
// NETWORK 1
//   _ManOn: Manual On
//   _ManOff: Manual Off
_rt1(CLK := _ManOn);
_ManOff R= _rt1.Q AND _ManOff;
IF _rt1.Q THEN _WarningNum := 0; END_IF
_rt2(CLK := _ManOff);
_ManOn R= _rt2.Q AND _ManOn;
IF _rt2.Q THEN _WarningNum := 0; END_IF

// NETWORK 2
_rt3(CLK := _AlarmMute);
IF _rt3.Q THEN _WarningNum := 0; END_IF

// NETWORK 3
//   Control.Inputs.AlarmMuteReset: Resets Alarm Mutes for all Alarms
_AlarmMute R= Control.Inputs.AlarmMuteReset;
END_METHOD

METHOD PRIVATE M_WarningMonitor
VAR_INPUT
END_VAR
VAR_INST
END_VAR
VAR_INST // added by the converter: edge detectors and wires of the graphical bodies
    _w1, _w2 : BOOL;
END_VAR
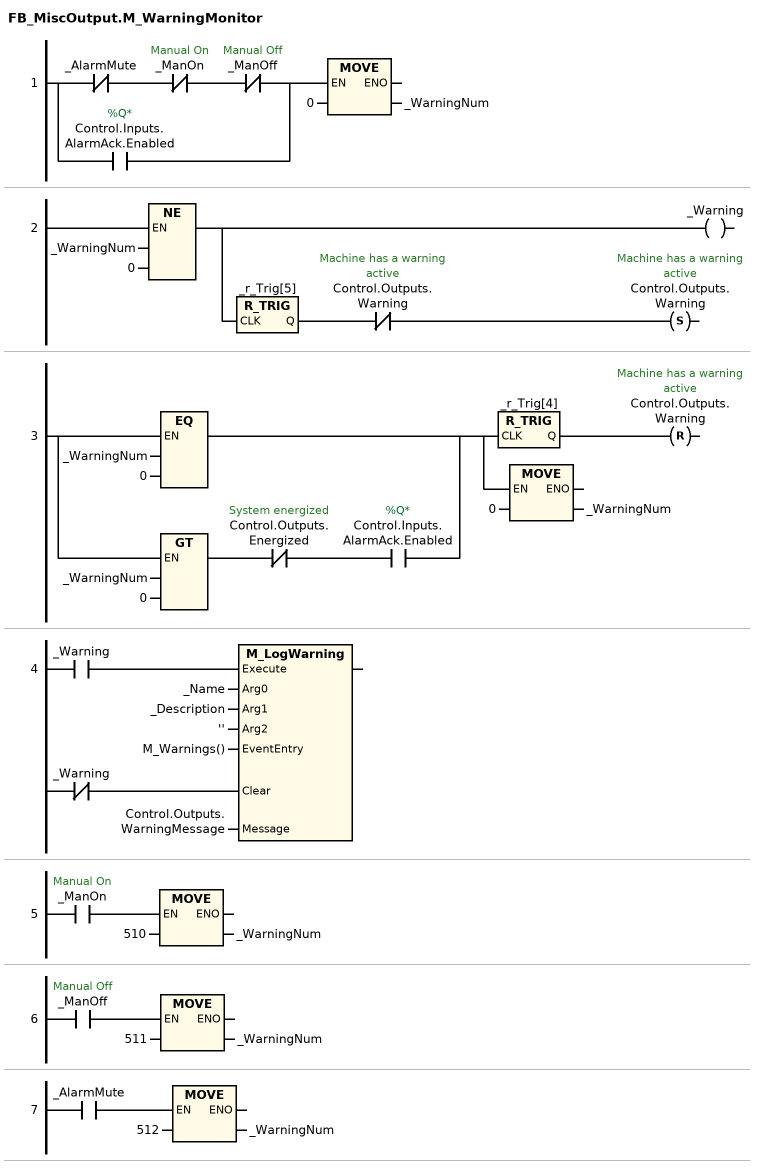
// NETWORK 1
//   _ManOn: Manual On
//   _ManOff: Manual Off
//   Control.Inputs.AlarmAck.Enabled: AT %Q*
IF NOT _AlarmMute AND NOT _ManOn AND NOT _ManOff OR Control.Inputs.AlarmAck.Enabled THEN _WarningNum := 0; END_IF

// NETWORK 2
//   Control.Outputs.Warning: Machine has a warning active
_w1 := _WarningNum <> 0;
_Warning := _w1;
_r_Trig[5](CLK := _w1); // R_TRIG
Control.Outputs.Warning S= _r_Trig[5].Q AND NOT Control.Outputs.Warning;

// NETWORK 3
//   Control.Outputs.Energized: System energized
//   Control.Inputs.AlarmAck.Enabled: AT %Q*
//   Control.Outputs.Warning: Machine has a warning active
_w2 := _WarningNum = 0 OR _WarningNum > 0 AND NOT Control.Outputs.Energized AND Control.Inputs.AlarmAck.Enabled;
_r_Trig[4](CLK := _w2); // R_TRIG
Control.Outputs.Warning R= _r_Trig[4].Q;
IF _w2 THEN _WarningNum := 0; END_IF

// NETWORK 4
M_LogWarning(Execute := _Warning, Arg0 := _Name, Arg1 := _Description, Arg2 := '', EventEntry := M_Warnings(), Clear := NOT _Warning, Message := Control.Outputs.WarningMessage);

// NETWORK 5
//   _ManOn: Manual On
IF _ManOn THEN _WarningNum := 510; END_IF

// NETWORK 6
//   _ManOff: Manual Off
IF _ManOff THEN _WarningNum := 511; END_IF

// NETWORK 7
IF _AlarmMute THEN _WarningNum := 512; END_IF
END_METHOD

METHOD PRIVATE M_Warnings : TcEventEntry
VAR_INPUT
END_VAR
CASE _WarningNum OF
	510: M_Warnings:= TC_Events.TcMiscOutput.W_510;//Manual ON
	511: M_Warnings:= TC_Events.TcMiscOutput.W_511;//Manual OFF		
	512: M_Warnings:= TC_Events.TcMiscOutput.W_512;//Alarm Mute Active						
ELSE
	M_Warnings:=  TC_Events.TcMiscOutput.W_Undefined;
END_CASE
END_METHOD

{attribute 'monitoring' := 'variable'}
PROPERTY PUBLIC ManOff : Bool
GET
ManOff := _ManOff;
END_GET
SET
_ManOff := ManOff;
END_SET
END_PROPERTY

{attribute 'monitoring' := 'variable'}
PROPERTY PUBLIC ManOn : Bool
GET
ManOn := _ManOn;
END_GET
SET
_ManOn := ManOn;
END_SET
END_PROPERTY

{attribute 'monitoring' := 'variable'}
PROPERTY PUBLIC Name : String[15]
GET
Name := _Name;
END_GET
SET
_Name := Name;
END_SET
END_PROPERTY

{attribute 'monitoring' := 'variable'}
PROPERTY PUBLIC OutputOff_ET : real
GET
OutputOff_ET := _OutputOff_ET;
END_GET
END_PROPERTY

{attribute 'monitoring' := 'variable'}
PROPERTY PUBLIC OutputOn_ET : real
GET
OutputOn_ET := _OutputOn_ET;
END_GET
END_PROPERTY

{attribute 'monitoring' := 'variable'}
PROPERTY PUBLIC StandbyReset : Bool
GET
StandbyReset := _ForceOff;
END_GET
SET
_ForceOff := StandbyReset;
END_SET
END_PROPERTY

{attribute 'monitoring' := 'variable'}
PROPERTY PUBLIC Value : Bool
GET
Value := _Value;
END_GET
SET
_Value := Value;
END_SET
END_PROPERTY

{attribute 'monitoring' := 'variable'}
PROPERTY PUBLIC Warning : Bool
GET
Warning := _Warning;
END_GET
END_PROPERTY

END_FUNCTION_BLOCK

// Objects/FB_OEE_V3_01/FB_OEE
FUNCTION_BLOCK FINAL FB_OEE
VAR_IN_OUT
	OEE									        : ST_OEE;
	OEE_SP									    : ST_OEE_SP;
	Control										: ST_System;
END_VAR
VAR
	_Current_Time								: ST_TIMEMANAGEMENT;
	_Current_Time_DT							: DATE_AND_TIME;
	_Current_Time_DW							: DWORD;
	_Pattern_Update								: BOOL;
	_Mach_Perf_Reset							: BOOL;
	_fb_MachinePerfomance						: FB_MachinePerformance;
	_riseEdge									: R_TRIG;
	_Start_Time_DT								: DATE_AND_TIME;
	_Length_Time_DT								: DATE_AND_TIME;
	_Operating_Time_DT							: DATE_AND_TIME;
	_Break_Time_DT								: DATE_AND_TIME;
	_Production_Time_DT							: DATE_AND_TIME;
	_Stop_Time_DT								: DATE_AND_TIME;
	_Start_Time_DW								: DWORD;
	_Length_Time_DW								: DWORD;
	_Stop_Time_DW								: DWORD;
	_Year_Month_Day_DT							: ARRAY [0..1] OF DATE_AND_TIME;
	_Year_Month_Day_TS							: ARRAY [0..1] OF TIMESTRUCT;
	_Year_Month_Day_DW							: ARRAY [0..1] OF DWORD;
	_Production_Time_T							: TIME;
	_Operating_Time_T							: TIME;
	_Break_Time_T								: TIME;
	_Production_Time_TS							: TIMESTRUCT;
	_Break_Time_TS								: TIMESTRUCT;
	_Operating_Time_TS							: TIMESTRUCT;
END_VAR


    _Current_Time.CurrentTime		:= (Control.SystemTime.CurrentTime);
    _Year_Month_Day_TS[0].wYear 	:= (Control.SystemTime.CurrentTime.wYear);
    _Year_Month_Day_TS[0].wMonth 	:= (Control.SystemTime.CurrentTime.wMonth);
    _Year_Month_Day_TS[0].wDay 		:= 1;
    _Year_Month_Day_TS[1].wYear 	:= (Control.SystemTime.CurrentTime.wYear);
    _Year_Month_Day_TS[1].wMonth    := (Control.SystemTime.CurrentTime.wMonth);
    _Year_Month_Day_TS[1].wDay 		:= 1;
    _Production_Time_TS.wYear 		:= (Control.SystemTime.CurrentTime.wYear);
    _Production_Time_TS.wMonth 		:= (Control.SystemTime.CurrentTime.wMonth);
    _Break_Time_TS.wYear 			:= (Control.SystemTime.CurrentTime.wYear);
    _Break_Time_TS.wMonth 			:= (Control.SystemTime.CurrentTime.wMonth);
    _Operating_Time_TS.wYear 		:= (Control.SystemTime.CurrentTime.wYear);
    _Operating_Time_TS.wMonth 		:= (Control.SystemTime.CurrentTime.wMonth);
    
    _riseEdge(CLK := OEE_SP.Active);
    OEE_SP.RisingEdge := _riseEdge.Q;
    
    IF (_riseEdge.Q) THEN
    	OEE_SP.Operating_Seconds := 0;
    	OEE_SP.Production_Seconds := 0;
    	OEE_SP.Break_Seconds := 0;
    	OEE_SP.SupplyDownTime_Seconds := 0;
    	OEE_SP.OutfeedDownTime_Seconds := 0;
    	OEE_SP.GoodPieces := 0;
    	OEE_SP.RejectPieces := 0;
		_Mach_Perf_Reset := TRUE;
	ELSE
		_Mach_Perf_Reset := FALSE;
    END_IF
    
    IF (_riseEdge.Q) OR (Control.SystemTime.MidnightPulse AND NOT OEE_SP.Active) THEN;
    	_Pattern_Update := TRUE;
    ELSE
    	_Pattern_Update := FALSE;
    END_IF
    
    IF _Pattern_Update THEN;  // Updates Start Year/Month/Day to Current and Length Year/Month/Day  @ Midnight Pulse @ Midnight Pulse
    	OEE_SP.Start.CurrentTime.wYear 	:= (Control.SystemTime.CurrentTime.wYear);
    	OEE_SP.Length.CurrentTime.wYear 	:= 0;	
    	OEE_SP.Start.CurrentTime.wMonth 	:= (Control.SystemTime.CurrentTime.wMonth);
    	OEE_SP.Length.CurrentTime.wMonth 	:= 0;
    	OEE_SP.Start.CurrentTime.wDay 	:= (Control.SystemTime.CurrentTime.wDay);
    	OEE_SP.Length.CurrentTime.wDay 	:= 0;
		OEE_SP.MachinePerformance[Control.PackMLState.CurrentState].Current_Time := 0;
		OEE_SP.MachinePerformance[Control.PackMLState.CurrentState].Current.CurrentTime.wHour := 0;
		OEE_SP.MachinePerformance[Control.PackMLState.CurrentState].Current.CurrentTime.wMinute := 0;
		OEE_SP.MachinePerformance[Control.PackMLState.CurrentState].Current.CurrentTime.wSecond := 0;
    END_IF

	//--------------------------------------------------------Stop Time Calculation---------------------------------------------------------
    _Start_Time_DT 			:= SYSTEMTIME_TO_DT(OEE_SP.Start.CurrentTime); 		// Converts Start Time format from TIMESTRUCT to DATE_AND_TIME
    _Length_Time_DT 		:= SYSTEMTIME_TO_DT(OEE_SP.Length.CurrentTime); 	// Converts Length Time format from TIMESTRUCT to DATE_AND_TIME
    _Year_Month_Day_DT[0] 	:= SYSTEMTIME_TO_DT(_Year_Month_Day_TS[0]);			// Year/Month TimeStuct for Calculation 		
    _Year_Month_Day_DT[1] 	:= SYSTEMTIME_TO_DT(_Year_Month_Day_TS[1]);			// Year/Month TimeStuct for Calculation
    _Start_Time_DW			:=DT_TO_DWORD(_Start_Time_DT); 						// Converts Start Time format from DATE_AND_TIME to DWORD for Calculation 
    _Length_Time_DW			:=DT_TO_DWORD(_Length_Time_DT); 					// Converts Length Time format from DATE_AND_TIME to DWORD for Calculation 
    _Year_Month_Day_DW[0]	:=DT_TO_DWORD(_Year_Month_Day_DT[0]); 				// Converts Year/Month Time format from DATE_AND_TIME to DWORD for Calculation 
    _Year_Month_Day_DW[1]	:=DT_TO_DWORD(_Year_Month_Day_DT[1]); 	       
                         
